E_AxisState.MOVE_ABS://-----------------------------------------------------------------------------------------MOVE_ABS:

							IF posTarget > fPositionLimitMin AND
							   posTarget < fPositionLimitMax
 								THEN 
									bReq_MoveABS := TRUE;
									eState := E_AxisState.MOVING_ABS;
							END_IF
							stY_Axis.bSetToHome			  :=FALSE;
							
							
E_AxisState.MOVING_ABS://-------------------------------------------------------------------------------------MOVING_ABS:

							IF fbMoveABS.Done THEN
									
									bReq_MoveABS := FALSE;
									eState := E_AxisState.IN_TARGET_POS;
									
							ELSIF tonMoveTimeout.Q THEN
									
									bReq_MoveABS := FALSE;
									eState := E_AxisState.ERROR;
							END_IF
							//TO KNOW POSITION OF AXIS
							GVL_HMI.bY_AxisInPosition1		:= FALSE;
							GVL_HMI.bY_AxisInPosition2		:= FALSE;
							GVL_HMI.bY_AxisInPosition3		:= FALSE;
							GVL_HMI.bY_AxisInHomePosition	:= FALSE;

E_AxisState.MOVE_REL:;
E_AxisState.MOVING_REL:;

E_AxisState.IN_TARGET_POS://-------------------------------------------------------------------------------IN_TARGET_POS:

							IF tonActionDone.Q THEN
								eState := E_AxisState.AXIS_READY;
							END_IF
							//TO KNOW THE POSITION OF THE AXIS
							IF stY_Axis.bSetToPosition[1] THEN
								GVL_HMI.bY_AxisInPosition1				:= TRUE;
							END_IF
							IF stY_Axis.bSetToPosition[2] THEN
								GVL_HMI.bY_AxisInPosition2				:= TRUE;
							END_IF
							IF stY_Axis.bSetToPosition[3] THEN
								GVL_HMI.bY_AxisInPosition3				:= TRUE;
							END_IF
							IF stY_Axis.bSetToHome THEN
								GVL_HMI.bY_AxisInHomePosition			:= TRUE;
							END_IF
E_AxisState.ERROR://-----------------------------------------------------------------------------------------------ERROR:

	 					eState := E_AxisState.ABORTED;
						
E_AxisState.MANUAL_MODE://-----------------------------------------------------------------------------------MANUAL_MODE:

							e_Manual();
					
							IF NOT CMD.bManualMode THEN
								eState := E_AxisState.ABORTED;
							END_IF

ELSE 
eState := E_AxisState.ABORTED;
END_CASE //------------------------------------------------------------------------------------------------------END_CASE

(******************************************************STATUS************************************************************)
// Module Status
status.bReady	:= eState = E_AxisState.AXIS_READY;

status.bBusy	:= eState <> E_AxisState.ABORTED	AND
				   eState <> E_AxisState.AXIS_READY AND
				   eState <> E_AxisState.IN_TARGET_POS AND
				   eState <> E_AxisState.ERROR;
				   
status.bDone	:= eState = E_AxisState.IN_TARGET_POS;

status.bError	:= eState = E_AxisState.ERROR OR 
				   fbPower.Error OR fbStop.Error OR fbMoveABS.Error OR fbMoveREL.Error; 
//---------------------------------------------------------------------------------------------------------------oldschoo1
END_ACTION

ACTION b_Call_AxisFBs:
// CTRL FBs Call

	fbPower 	(Axis:=refY_Axis, Enable:=bReq_Power, Enable_Positive:=bReq_Power, Enable_Negative:=bReq_Power);
	fbReset 	(Axis:=refY_Axis, Execute:=bReq_Reset);
	
  fbMoveABS 	(Axis:=refY_Axis, Execute:=bReq_MoveABS, 
				 Position:=posTarget, Velocity:= SEL(bRetract,cfgAxis.fTargetVelocity,cfgAxis.fRetractVelocity));
  fbMoveREL 	(Axis:=refY_Axis, Execute:=FALSE);
 	 fbStop 	(Axis:=refY_Axis, Execute:=FALSE);
  fbReadPos		(Axis:=refY_Axis, Enable:=eState=E_AxisState.HOMING);
fbParameter[0]  (Axis:=refY_Axis, Enable:=TRUE, ParameterNumber:=MC_AXISPARAMETER.AxisMinSoftPosLimit, Value=>fLimitPositionLow);
fbParameter[1]  (Axis:=refY_Axis, Enable:=TRUE, ParameterNumber:=MC_AXISPARAMETER.AxisMaxSoftPosLimit, Value=>fLimitPositionHigh);
fbReadStatus	(Axis:=refY_Axis, Enable:=TRUE, Status=>stAxisStatus, Error=>bAxisInError);
//-----------------------------------------------------------------------------------------------------------------------oldschoo1
END_ACTION

METHOD c_Get_TargetPositon	:LREAL
VAR_INPUT

	// Positions
    posHome     			:LREAL;
    posPoints   			:ARRAY[1..3]OF LREAL;
    fOffsets  				:ARRAY[1..3]OF LREAL;
	
	// Set Target Flags
    bSetHome    			:BOOL;
    bSetPoint   			:ARRAY[1..3]OF BOOL;
	
END_VAR
//----------------------------------------------------------oldschoo1


VAR
	idx           			:INT;
	posTargeteBase	     	:LREAL;
END_VAR
IF bSetHome THEN
    		posTargeteBase := posHome;
ELSE
	
			FOR idx:= 1 TO 3 
			DO
					IF bSetPoint[idx] THEN
						posTargeteBase := posPoints[idx] + fOffsets[idx];
						EXIT;
					END_IF		
			END_FOR
END_IF

c_Get_TargetPositon	:= posTargeteBase;
//--------------------------------------------------------------oldschoo1
END_METHOD

ACTION d_Get_CurrentPosition:
IF fbReadPos.Valid THEN fCurrentPosition:=fbReadPos.Position; END_IF
//----------------------------------------------------------oldschoo1
END_ACTION

ACTION e_Manual:
posTarget := c_Get_TargetPositon(
															posHome 	:= cfgAxis.posHome,
															posPoints   := cfgAxis.posWorkPositions,
															fOffsets	:= fOffsets,
															bSetHome 	:= stY_Axis.bSetToHome,
															bSetPoint 	:= stY_Axis.bSetToPosition
															);	
trigbMoveToPos( CLK := GVL_HMI.bMoveToPos );
IF GVL_HMI.bY_AxisPosition1 THEN
	stY_Axis.bSetToPosition[1]			:= TRUE;
	GVL_HMI.bMoveToPos					:= TRUE;
END_IF
IF GVL_HMI.bY_AxisPosition2 THEN
	stY_Axis.bSetToPosition[2]			:= TRUE;
	GVL_HMI.bMoveToPos					:= TRUE;
END_IF
IF GVL_HMI.bY_AxisPosition3 THEN
	stY_Axis.bSetToPosition[3]			:= TRUE;
	GVL_HMI.bMoveToPos					:= TRUE;
END_IF
IF GVL_HMI.bY_HomePosition THEN
	stY_Axis.bSetToHome					:= TRUE;
	GVL_HMI.bMoveToPos					:= TRUE;
END_IF
	
IF trigbMoveToPos.Q THEN
	nManualModeState					:=10;
END_IF

CASE nManualModeState OF
	
10:
IF posTarget > fPositionLimitMin AND
		posTarget < fPositionLimitMax THEN 
		bReq_MoveABS 					:= TRUE;
		GVL_HMI.bY_AxisInPosition1Man	:= FALSE;
		GVL_HMI.bY_AxisInPosition2Man	:= FALSE;
		GVL_HMI.bY_AxisInPosition3Man	:= FALSE;
		GVL_HMI.bY_AxisInHomePositionMan:= FALSE;
		nManualModeState				:=20;
	END_IF	
20:
IF fbMoveABS.Done THEN	
	IF stY_Axis.bSetToPosition[1] THEN
		GVL_HMI.bY_AxisInPosition1Man	:= TRUE;
	END_IF
	IF stY_Axis.bSetToPosition[2] THEN
		GVL_HMI.bY_AxisInPosition2Man	:= TRUE;
	END_IF
	IF stY_Axis.bSetToPosition[3] THEN
		GVL_HMI.bY_AxisInPosition3Man	:= TRUE;
	END_IF
	IF stY_Axis.bSetToHome THEN
		GVL_HMI.bY_AxisInHomePositionMan:= TRUE;
	END_IF
	nManualModeState					:=30;
END_IF
	
30:								
		bReq_MoveABS 					:= FALSE;
		stY_Axis.bSetToPosition[1]		:= FALSE;
		stY_Axis.bSetToPosition[2]		:= FALSE;
		stY_Axis.bSetToPosition[3]		:= FALSE;
		stY_Axis.bSetToHome				:= FALSE;
		GVL_HMI.bMoveToPos				:= FALSE;
		
IF NOT GVL_Master.stMachineStatus.bManualMode THEN
		GVL_HMI.bY_AxisInPosition1Man	:= FALSE;
		GVL_HMI.bY_AxisInPosition2Man	:= FALSE;
		GVL_HMI.bY_AxisInPosition3Man	:= FALSE;
		GVL_HMI.bY_AxisInHomePositionMan:= FALSE;
END_IF
END_CASE
END_ACTION

END_PROGRAM

// ---- POUs/01_MODULES/KISTLER/K_Master_Kistler.TcPOU
PROGRAM K_Master_Kistler
VAR
	
	bFirstRun							:BOOL:=TRUE;
	
	//Module CTRL
	eState								:E_KistlerState:=E_KistlerState.ENABLE_PLC_CTRL;
	eErrorID							:E_KistlerErrorID;
	
	//Parameters
	fHomePositionTolerance				:REAL:= 1.5;	// > 2mm may cause Pack insertion issues
	fbForceMonitor						:FB_ForceMonitor;
	FBDistanceMonitor					: FB_DistanceMonitor;
	fUVT_00								:REAL;
	fUVT_01								:REAL;	
	fDistanceSetpoint					:REAL;
	//Timers && Triggers
	tonAbortModule						:Tc2_Standard.TON;
	tonResetError						:Tc2_Standard.TON;
	tonEnableDrive						:Tc2_Standard.TON;
	tonActionDone						:Tc2_Standard.TON;
	tonActionTimeout					:Tc2_Standard.TON;
	tonPowerUpTimeout					:Tc2_Standard.TON;	
	tonDelaySignals						:ARRAY[1..11]OF Tc2_Standard.TON;
	
	rcmdbExecute						:R_TRIG;
	
	//EtherCAT - Kistler CTRL
	stSendCMD							:ST_KistlerData_CMD;
	

	//Com Data Proccessing
	stTemp								:ST_KistlerData_Temporary;//Temp. only
	fbUnpack							:ARRAY[0..199]OF FB_UnpackByteToBoolArray;
	fbByte2Real							:FB_ArrayOfByte2Real;
	fbRealPosition2Byte					:FB_Real2ArrayOfByte;
	fbRealSpeed2Byte					:FB_Real2ArrayOfByte;
	fbPositiontosend					:FB_Byte_To_Bits;
	fbSpeedtosend						:FB_Byte_To_Bits;
	
	// Live readings Local
	rKistlerLive_X						:REAL;	//Travel
	rKistlerLive_Y						:REAL;	//Force
	
	// Process Record
	bForceMonitorActive					:BOOL;	//Recording Start/Stop
	
	
	//Support variables
	idx1								:INT;	//indexer
	idx2								:INT;	//indexer
	idx3								:INT;	//indexer
	
	//Manual
	trigCycleMan						:R_TRIG;
	tonRstCycSignalMan					:TON;
	bTest								:BOOL;
	
	rPosition							:FB_BytesToReal;
	rSpeed								:FB_BytesToReal;
	
	bDistancePass						: BOOL;
	bDistanceFail						: BOOL;
	
END_VAR
VAR_OUTPUT
	stKistlerReport						:ST_ProcessReport;
END_VAR


//--------------------IN/OUT-----------------------------------------------------------------*
VAR_INPUT	
	CMD									:ST_ModuleCMD;	
END_VAR
VAR_OUTPUT	
	STATUS								:ST_ModuleStatus;
	stReceived							:ST_KistlerData_Status;	
END_VAR
//-----------------------------------------------------------------------------------oldschoo1

PRG_Fault_Kistler(aAlarms := GVL_Master.stAlarms);
//Call for Actions
a_Unpack_Received();
b_Ctrl_Kistler();
d_Monitor_ProcessForce();
f_Pack_DataToSend();


// Map to HMI
GVL_HMI.rKistlerLiveReading_X		:= rKistlerLive_X;	//Realtime X travel distance
GVL_HMI.rKistlerLiveReading_Y		:= rKistlerLive_Y;	//Realtime Y force reading

fDistanceSetpoint				:= GVL_PERSISTENT.rReservoir_BottomPosition - GVL_PERSISTENT.rReservoir_Bottomlimitoffset;

//--------------------------------------------------------------------------oldschoo1

ACTION a_Unpack_Received:
//Thanks for the Telegram, it's been received:)
FOR idx1:= 0 TO 199 
DO 
fbUnpack[idx1].inputByte := GVL_MODULES.stKistler.st_TelegramDataIn[idx1];
fbUnpack[idx1](outputBits := stTemp.arrInBits[idx1]);
END_FOR
//---------------------------------------------------------------oldschoo1

//  Byte 0  –  Basic CTRL Mirror  ---------------------------------------
stReceived.bStart_Mirror						:= stTemp.arrInBits[0][0];
stReceived.bTareY_Mirror						:= stTemp.arrInBits[0][1];
stReceived.bZeroX_Mirror						:= stTemp.arrInBits[0][2];
stReceived.bSTestX_Mirror						:= stTemp.arrInBits[0][3];
stReceived.bSTestY_Mirror						:= stTemp.arrInBits[0][4];
stReceived.bMasterMeas_Mirror					:= stTemp.arrInBits[0][6];
stReceived.bIncZero_Mirror						:= stTemp.arrInBits[0][7];

//  Byte 1  –  Login Mirror  --------------------------------------------
stReceived.bAckAdminGlobal_Mirror				:= stTemp.arrInBits[1][0];
stReceived.bAckAdmin_Mirror						:= stTemp.arrInBits[1][1];
stReceived.bAccess_Mirror						:= stTemp.arrInBits[1][3];
stReceived.bAuto_Mirror							:= stTemp.arrInBits[1][4];
stReceived.bStatReset_Mirror					:= stTemp.arrInBits[1][5];
stReceived.bStatDisable_Mirror					:= stTemp.arrInBits[1][6];
stReceived.bTareExtY_Mirror						:= stTemp.arrInBits[1][7];

//  Byte 2  –  Measurement Program No. Mirror  --------------------------
stReceived.mpNumber_Mirror[0]					:= stTemp.arrInBits[2][0];
stReceived.mpNumber_Mirror[1]					:= stTemp.arrInBits[2][1];
stReceived.mpNumber_Mirror[2]					:= stTemp.arrInBits[2][2];
stReceived.mpNumber_Mirror[3]					:= stTemp.arrInBits[2][3];
stReceived.mpNumber_Mirror[4]					:= stTemp.arrInBits[2][4];
stReceived.mpNumber_Mirror[5]					:= stTemp.arrInBits[2][5];
stReceived.mpNumber_Mirror[6]					:= stTemp.arrInBits[2][6];

//  Byte 3  –  Service / Brake  -----------------------------------------
stReceived.bResetSNGen_Mirror					:= stTemp.arrInBits[3][2];
stReceived.bBrakeTestActive						:= stTemp.arrInBits[3][5];
stReceived.bExportPvt_Mirror					:= stTemp.arrInBits[3][6];

//  Byte 4  –  Configurable Inputs Mirror  ------------------------------
stReceived.bIUni_Mirror[0]						:= stTemp.arrInBits[4][0];
stReceived.bIUni_Mirror[1]						:= stTemp.arrInBits[4][1];
stReceived.bIUni_Mirror[2]						:= stTemp.arrInBits[4][2];
stReceived.bIUni_Mirror[3]						:= stTemp.arrInBits[4][3];
stReceived.bIUni_Mirror[4]						:= stTemp.arrInBits[4][4];
stReceived.bIUni_Mirror[5]						:= stTemp.arrInBits[4][5];
stReceived.bIUni_Mirror[6]						:= stTemp.arrInBits[4][6];
stReceived.bIUni_Mirror[7]						:= stTemp.arrInBits[4][7];

//  Byte 6  –  Global Status  -------------------------------------------
stReceived.bReady								:= stTemp.arrInBits[6][0];
stReceived.bOkTotal								:= stTemp.arrInBits[6][1];
stReceived.bNokTotal							:= stTemp.arrInBits[6][2];
stReceived.bNoPass								:= stTemp.arrInBits[6][3];
stReceived.bWarning								:= stTemp.arrInBits[6][6];
stReceived.bAlarm								:= stTemp.arrInBits[6][7];

//  Byte 7  –  Switching Signals  ---------------------------------------
stReceived.bS1									:= stTemp.arrInBits[7][0];
stReceived.bS2									:= stTemp.arrInBits[7][1];

//  Byte 8  –  O_UNI  ---------------------------------------------------
stReceived.bO_UNI[0]							:= stTemp.arrInBits[8][0];
stReceived.bO_UNI[1]							:= stTemp.arrInBits[8][1];

//  Byte 9  –  Drive / Sequence Mirror  ---------------------------------
stReceived.bDriveEnable_Mirror					:= stTemp.arrInBits[9][0];
stReceived.bRunSequence_Mirror					:= stTemp.arrInBits[9][1];
stReceived.bDriveHome_Mirror					:= stTemp.arrInBits[9][2];
stReceived.bDriveRef_Mirror						:= stTemp.arrInBits[9][3];
stReceived.bJogFwd_Mirror						:= stTemp.arrInBits[9][4];
stReceived.bJogBack_Mirror						:= stTemp.arrInBits[9][5];
stReceived.bWaitRequest							:= stTemp.arrInBits[9][6];
stReceived.bBrakeTestDone						:= stTemp.arrInBits[9][7];

//  Byte 10 –  Sequence State  -------------------------------------------
stReceived.bSeqStopped							:= stTemp.arrInBits[10][0];
stReceived.bSeqEnd								:= stTemp.arrInBits[10][1];
stReceived.bOnlineEoNok							:= stTemp.arrInBits[10][2];
stReceived.bSeqExtStop							:= stTemp.arrInBits[10][3];
stReceived.bSeqError							:= stTemp.arrInBits[10][4];
stReceived.bDriveEnabled						:= stTemp.arrInBits[10][5];
stReceived.bHomePosReached						:= stTemp.arrInBits[10][6];
stReceived.bRefPosReached						:= stTemp.arrInBits[10][7];

//  Byte 11 –  Servo / Safety  -------------------------------------------
stReceived.bStandstill							:= stTemp.arrInBits[11][0];
stReceived.bBrakeTestReq						:= stTemp.arrInBits[11][1];
stReceived.bServoWarn							:= stTemp.arrInBits[11][2];
stReceived.bServoError							:= stTemp.arrInBits[11][3];
stReceived.bSMES_Or_STO							:= stTemp.arrInBits[11][4];
stReceived.bSMST2								:= stTemp.arrInBits[11][5];
stReceived.bSMM1								:= stTemp.arrInBits[11][6];
stReceived.bUserModeActive						:= stTemp.arrInBits[11][7];

//  Byte 12 –  Current Sequence Mirror  ----------------------------------
stReceived.bCurrSeqMain_Mirror					:= stTemp.arrInBits[12][0];
stReceived.bCurrSeqSub_Mirror					:= stTemp.arrInBits[12][1];

//  Byte 19 –  Device / Transfer Flags  ----------------------------------
stReceived.bTransmissionFault					:= stTemp.arrInBits[19][0];
stReceived.bAck									:= stTemp.arrInBits[19][1];
stReceived.bDeviceAvailable						:= stTemp.arrInBits[19][2];
stReceived.bMpChanged							:= stTemp.arrInBits[19][4];
stReceived.bGlobalChanged						:= stTemp.arrInBits[19][6];
stReceived.bBackupComplete						:= stTemp.arrInBits[19][7];

(************************************Payload**************************************)
//  Bytes 20-27 –  Live XY values  ----------------------------------------------*
FOR idx3:= 20 TO 23					
DO
stReceived.pvCurrentValueX[idx3] := FUN_PackBoolArrayToByte(stTemp.arrInBits[idx3]);
																		    END_FOR
							     fbByte2Real.arrBytes := stReceived.pvCurrentValueX;
							     fbByte2Real();rKistlerLive_X := fbByte2Real.rValue;
																			
FOR idx3:= 24 TO 27					
DO
stReceived.pvCurrentValueY[idx3] := FUN_PackBoolArrayToByte(stTemp.arrInBits[idx3]);
																			END_FOR
							     fbByte2Real.arrBytes := stReceived.pvCurrentValueY;
							     fbByte2Real();rKistlerLive_Y := fbByte2Real.rValue;
//--------------------------------------------------------------------------oldschoo1

rPosition(inBytes:= , outReal=> );
rSpeed(inBytes:= , outReal=> );
END_ACTION

ACTION b_Ctrl_Kistler:
// Timmers && Triggers
tonActionDone     (IN:= FALSE,
			       PT:= T#100MS);
tonActionTimeout  (IN:= eState=E_KistlerState.WAIT_CYCLE_DONE,
			       PT:= T#90S);
tonPowerUpTimeout (IN:= eState=E_KistlerState.ENABLE_DRIVE,
				   PT:=T#20S);				   
tonResetError     (IN:= stReceived.bServoError OR stReceived.bAlarm,
			       PT:= T#500MS);
tonAbortModule	  (IN:= cmd.bAbort OR (NOT stSafety.bSafety_OK) OR (NOT cmd.bEnable),
				   PT:= T#100MS);
				   
//Signal pulses && delays				  
tonDelaySignals[1](IN:= eState=E_KistlerState.ENABLE_PLC_CTRL AND stSendCMD.bAckAdminGlobal,
				   PT:= T#100MS);
tonDelaySignals[2](IN:= eState=E_KistlerState.RESET_ERROR AND (stReceived.bAlarm OR stReceived.bServoError) AND NOT tonDelaySignals[3].Q,
				   PT:= T#1S);
tonDelaySignals[3](IN:= eState=E_KistlerState.RESET_ERROR AND stSendCMD.bAckAdmin,
				   PT:= T#1S);
tonDelaySignals[4](IN:= eState=E_KistlerState.ENABLE_DRIVE,
				   PT:= T#100MS);
tonDelaySignals[5](IN:= eState=E_KistlerState.SET_PARAMETERS,
				   PT:=T#330MS);
tonDelaySignals[6](IN:=eState=E_KistlerState.RECORD_CYCLE_DATA, 
				   PT:=T#50MS);				   
tonDelaySignals[7](IN:=eState=E_KistlerState.ERROR, 
				   PT:=T#330MS);
tonDelaySignals[8](IN:=eState=E_KistlerState.PRESS_CYCLE, 
				   PT:=T#330MS);
tonDelaySignals[9](IN:=eState=E_KistlerState.GOTO_HOME_POS, 
				   PT:=T#330MS);
tonDelaySignals[10](IN:=eState=E_KistlerState.SET_PARAMETERS AND stReceived.bTareY_Mirror AND tonDelaySignals[5].Q, 
				   PT:=T#3S);
tonDelaySignals[11]( IN := NOT stReceived.bAlarm, PT := T#1S);

rcmdbExecute( CLK := cmd.bExecute);
(*****************************************************RESET**********************************************************)
// Reset Errors
(*IF cmd.bReset OR tonResetError.Q THEN
 			  
			status.bError 	:= TRUE;
            eState := E_KistlerState.RESET_ERROR;
			END_IF*)

// Abort Action
IF tonAbortModule.q THEN
	
			stSendCMD.bDriveEnable	:= FALSE;
			stSendCMD.bAckAdmin		:= FALSE;
			stSendCMD.bDriveToRef	:= FALSE;
			stSendCMD.bTareY 		:= FALSE;
			stSendCMD.bRunSequence  := FALSE;
			eState := E_KistlerState.ABORTED;
			END_IF	
(*******************************************************CTRL**********************************************************)
IF CMD.bManualMode THEN
	eState := E_KistlerState.MANUAL;
END_IF
// Kistler CTRL State Machine
CASE eState OF //-----------------------------------------------------------------------------------------------------SM

E_KistlerState.ENABLE_PLC_CTRL://-----------------------------------------------------------------------ENABLE_PLC_CTRL:

						IF stReceived.bReady AND NOT bSystemPoweringUP THEN
								stSendCMD.bAuto:=TRUE; 
						ELSIF NOT stReceived.bReady THEN
								status.nErrorID:= TO_INT(eErrorID=E_KistlerErrorID.COMUNICATION_ERROR);
						END_IF
								
						IF stReceived.bAuto_Mirror THEN
								stSendCMD.bAckAdminGlobal:=TRUE;
						END_IF
						IF tonDelaySignals[1].Q THEN
 								stSendCMD.bAckAdminGlobal:=FALSE;
								eState := E_KistlerState.ABORTED;
								END_IF

E_KistlerState.ABORTED://---------------------------------------------------------------------------------------ABORTED:
					
						IF (NOT stReceived.bAuto_Mirror) AND 
						   (NOT cmd.bAbort) AND stSafety.bSafety_OK AND cmd.bEnable THEN
								eState := E_KistlerState.ENABLE_PLC_CTRL;
							
						ELSIF stReceived.bAuto_Mirror AND 
							 (NOT cmd.bAbort) AND stSafety.bSafety_OK AND cmd.bEnable THEN
								eState := E_KistlerState.ENABLE_DRIVE;
						END_IF
								

E_KistlerState.ENABLE_DRIVE://-----------------------------------------------------------------------------ENABLE_DRIVE:
	
						c_Select_Program();

						IF tonDelaySignals[4].Q THEN
								stSendCMD.bDriveEnable:=TRUE; END_IF
						
						IF stReceived.bDriveEnabled THEN
								eState := E_KistlerState.RESET_ERROR;
								
						ELSIF (NOT stReceived.bDriveEnabled) AND tonPowerUpTimeout.Q THEN
								status.nErrorID:= TO_INT(eErrorID=E_KistlerErrorID.ENABLE_DRIVE_ERROR);
								eState := E_KistlerState.ERROR;
						END_IF

E_KistlerState.RESET_ERROR://-------------------------------------------------------------------------------RESET_ERROR:
					
						IF stReceived.bAlarm OR stReceived.bServoError  THEN
								IF tonDelaySignals[2].Q THEN
								stSendCMD.bAckAdmin:=TRUE; END_IF
						END_IF
		
						IF tonDelaySignals[3].Q THEN
								stSendCMD.bAckAdmin:=FALSE; END_IF
								
						IF (tonDelaySignals[11].Q) AND (NOT stReceived.bServoError) THEN
								stSendCMD.bAckAdmin:=FALSE;
								status.nErrorID:= TO_INT(eErrorID=E_KistlerErrorID.NO_ERROR);
								eState := E_KistlerState.GOTO_HOME_POS;
						END_IF
						
E_KistlerState.GOTO_HOME_POS://---------------------------------------------------------------------------GOTO_HOME_POS:

						IF NOT stReceived.bHomePosReached AND stReceived.bReady AND
								tonDelaySignals[9].Q THEN

								stSendCMD.bDriveToRef:= TRUE;
						END_IF
						
						IF stReceived.bHomePosReached OR rKistlerLive_X < fHomePositionTolerance THEN

								stSendCMD.bDriveToRef:= FALSE;
								eState := E_KistlerState.SET_PARAMETERS;
						END_IF
	
E_KistlerState.SET_PARAMETERS://-------------------------------------------------------------------------SET_PARAMETERS:

						stSendCMD.bTareY := TRUE;
						fUVT_00:= GVL_PERSISTENT.rReservoir_BottomPosition;
						fUVT_01:= GVL_PERSISTENT.rKistlerForce_Speed;
						
						IF stReceived.bTareY_Mirror AND tonDelaySignals[5].Q THEN
								stSendCMD.bTareY := FALSE;
								eState := E_KistlerState.PRESS_READY;
						END_IF

E_KistlerState.PRESS_READY://-------------------------------------------------------------------------------PRESS_READY:

						IF stReceived.bReady AND rcmdbExecute.Q THEN
								eState := E_KistlerState.PRESS_CYCLE;
						END_IF

						
E_KistlerState.PRESS_CYCLE://-------------------------------------------------------------------------------PRESS_CYCLE:


						stSendCMD.bRunSequence := TRUE;
						
						IF stReceived.bRunSequence_Mirror  AND tonDelaySignals[8].Q THEN
								eState := E_KistlerState.WAIT_CYCLE_DONE;
						END_IF
						
E_KistlerState.WAIT_CYCLE_DONE://-----------------------------------------------------------------------WAIT_PRESS_DONE:
						
						IF stReceived.bSeqEnd AND NOT stReceived.bSeqError THEN

								stSendCMD.bRunSequence := FALSE;	
								eState := E_KistlerState.RECORD_CYCLE_DATA;
						
						ELSIF stReceived.bSeqError THEN
								status.nErrorID:= TO_INT(eErrorID=E_KistlerErrorID.PROCESS_ERROR);
								eState := E_KistlerState.ERROR;
	
						ELSIF tonActionTimeout.Q THEN
								status.nErrorID:= TO_INT(eErrorID=E_KistlerErrorID.ACTION_TIMEOUT_ERROR);
								eState := E_KistlerState.ERROR;		
						END_IF
					
E_KistlerState.RECORD_CYCLE_DATA://-------------------------------------------------------------------RECORD_CYCLE_DATA:

			 			

			stKistlerReport.bKis_Pass := fbForceMonitor.bPass AND bDistancePass;
			stKistlerReport.bKis_Fail := fbForceMonitor.bFail OR bDistanceFail;
			stKistlerReport.rKis_HighestRecordedForce := fbForceMonitor.fHighestRecordedForce;
			stKistlerReport.rKis_LowestRecordedForce := fbForceMonitor.fLowestRecordedForce;
			stKistlerReport.rKis_DistanceRecord:=FBDistanceMonitor.MaxDistance;
			stKistlerReport.rKis_Settings_ForceUPPERtreshold := GVL_PERSISTENT.rKistlerForce_UpperLimit;
			stKistlerReport.rKis_Settings_ForceLOWERtreshold := GVL_PERSISTENT.rKistlerForce_LowerLimit;
			stKistlerReport.rKis_Settings_StartMeasurePoint := GVL_PERSISTENT.rReservoir_ContactPosition;
			stKistlerReport.rKis_Settings_ReservoirBottomPoint := GVL_PERSISTENT.rReservoir_BottomPosition;
			
						IF tonDelaySignals[6].Q THEN
								eState := E_KistlerState.PRESS_READY; END_IF	
				
E_KistlerState.JOG_MODE:;
E_KistlerState.ERROR://-------------------------------------------------------------------------------------------ERROR:
						stSendCMD.bDriveEnable	:= FALSE;
						stSendCMD.bAckAdmin		:= FALSE;
						stSendCMD.bDriveToRef	:= FALSE;
						stSendCMD.bTareY 		:= FALSE;
						stSendCMD.bRunSequence  := FALSE;
						
						IF tonDelaySignals[7].Q THEN
					 			eState := E_KistlerState.ABORTED; END_IF
E_KistlerState.MANUAL:
						g_Manual();
						IF NOT CMD.bManualMode THEN
							eState := E_KistlerState.ABORTED;
						END_IF
								
ELSE 
eState := E_KistlerState.ABORTED;
END_CASE //-----------------------------------------------------------------------------------------------------END_CASE

// -------------------------------------------HMI Show Record -------------------------------------------------------//
				IF 	eState = E_KistlerState.PRESS_READY AND (stKistlerReport.bKis_Pass OR stKistlerReport.bKis_Fail) THEN 
					
					GVL_HMI.rKisterldistanceHMI:= FBDistanceMonitor.MaxDistance;
					GVL_HMI.rKisterlForceHMI:=stKistlerReport.rKis_HighestRecordedForce;
					ELSE 
						GVL_HMI.rKisterldistanceHMI:= GVL_HMI.rKistlerLiveReading_X;
						GVL_HMI.rKisterlForceHMI:= GVL_HMI.rKistlerLiveReading_Y;
					END_IF


(******************************************************STATUS***********************************************************)
// Module Status
status.bReady				:= eState = E_KistlerState.PRESS_READY AND 
							   			stReceived.bReady;

status.bBusy				:= eState <> E_KistlerState.ABORTED		AND
				   			   eState <> E_KistlerState.PRESS_READY AND
				   			   eState <> E_KistlerState.ERROR;
				   
status.bActionInProggress	:= eState = E_KistlerState.PRESS_CYCLE OR
				   			   eState = E_KistlerState.WAIT_CYCLE_DONE OR
							   eState = E_KistlerState.RECORD_CYCLE_DATA;
							   
status.bDone				:= eState = E_KistlerState.RECORD_CYCLE_DATA;

status.bError				:= eState = E_KistlerState.ERROR OR 
				   			   stReceived.bServoError; 				 
//-------------------------------------------------------------------------------------------------------------oldschoo1
END_ACTION

ACTION c_Select_Program:
// MP No.selection is 6-bits binary
stSendCMD.mpNumber[0]:=1;  
stSendCMD.mpNumber[1]:=1;  
stSendCMD.mpNumber[2]:=0;  
stSendCMD.mpNumber[3]:=0;  
stSendCMD.mpNumber[4]:=0;  
stSendCMD.mpNumber[5]:=0;  
stSendCMD.mpNumber[6]:=0; 
//------------------------oldschoo1
END_ACTION

ACTION d_Monitor_ProcessForce:

//Trigger
bForceMonitorActive := (eState=E_KistlerState.PRESS_CYCLE OR eState=E_KistlerState.WAIT_CYCLE_DONE);(*AND 
					   (rKistlerLive_X > GVL_PERSISTENT.rReservoir_ContactPosition AND
						rKistlerLive_X < GVL_PERSISTENT.rReservoir_BottomPosition) AND stReceived.bO_UNI[0]*);

//Monitor
fbForceMonitor(
				bEnable := eState=E_KistlerState.PRESS_CYCLE OR eState=E_KistlerState.WAIT_CYCLE_DONE
							OR eState = E_KistlerState.RECORD_CYCLE_DATA,//stReceived.bAuto_Mirror,
				bActive := bForceMonitorActive,
				bReset	:= eState=E_KistlerState.PRESS_READY OR 
						   eState=E_KistlerState.ERROR OR cmd.bReset,
				fDistanceSetpoint := fDistanceSetpoint,
				fDistance := rKistlerLive_X,
 
				fForceInput 		  := rKistlerLive_Y,
				bPass				  =>,
				bFail				  =>,
				fHighestRecordedForce =>,
				fLowestRecordedForce  =>,
				fThreshold_UpperLimit := GVL_PERSISTENT.rKistlerForce_UpperLimit,
				fThreshold_LowerLimit := GVL_PERSISTENT.rKistlerForce_LowerLimit,
				fDebounceTolerance	  := GVL_PERSISTENT.rMeasurementTolerance );
				
//------------------------------------------------------------------------------------------------oldschoo1


FBDistanceMonitor(
	StartSignal:= eState=E_KistlerState.PRESS_CYCLE , 
	EndSignal:= stReceived.bSeqEnd,//eState=E_KistlerState.PRESS_READY, 
	DistanceMaxSetpoint:= , 
	DistanceInput:= rKistlerLive_X,
	fDistanceSetpoint := fDistanceSetpoint, 
	MaxDistance=> , 
	IsMeasuring=>,
	bDistancePass =>bDistancePass,
	bDistanceFail => bDistanceFail);
END_ACTION

ACTION f_Pack_DataToSend:
//  Byte 0  –  Basic CTRL  ----------------------------------------------*
stTemp.arrOutBits[0][0] 					:= stSendCMD.bStart;
stTemp.arrOutBits[0][1] 					:= stSendCMD.bTareY;
											   stSendCMD.bZeroX:=0; //Carefull, Teach Global 0 Position!!!
stTemp.arrOutBits[0][2] 					:= stSendCMD.bZeroX;//*
stTemp.arrOutBits[0][3] 					:= stSendCMD.bSTestX;
stTemp.arrOutBits[0][4] 					:= stSendCMD.bSTestY;
stTemp.arrOutBits[0][5] 					:= 0;
stTemp.arrOutBits[0][6] 					:= stSendCMD.bMasterMeas;
stTemp.arrOutBits[0][7] 					:= stSendCMD.bIncZero;
//  Byte 1  –  Login / Mode  ---------------------------------------------*
stTemp.arrOutBits[1][0] 					:= stSendCMD.bAckAdminGlobal;
stTemp.arrOutBits[1][1] 					:= stSendCMD.bAckAdmin;
stTemp.arrOutBits[1][2] 					:= 0;
stTemp.arrOutBits[1][3] 					:= stSendCMD.bAccess;
stTemp.arrOutBits[1][4] 					:= stSendCMD.bAuto;		//Set false to use TeachingPendant
stTemp.arrOutBits[1][5] 					:= stSendCMD.bStatReset;
stTemp.arrOutBits[1][6] 					:= stSendCMD.bStatDisable;
stTemp.arrOutBits[1][7] 					:= stSendCMD.bTareExtY;
//  Byte 2  –  Measurement Program No.  ----------------------------------*
stTemp.arrOutBits[2][0] 					:= stSendCMD.mpNumber[0];  
stTemp.arrOutBits[2][1] 					:= stSendCMD.mpNumber[1];
stTemp.arrOutBits[2][2] 					:= stSendCMD.mpNumber[2];
stTemp.arrOutBits[2][3] 					:= stSendCMD.mpNumber[3];
stTemp.arrOutBits[2][4] 					:= stSendCMD.mpNumber[4];
stTemp.arrOutBits[2][5] 					:= stSendCMD.mpNumber[5];
stTemp.arrOutBits[2][6] 					:= stSendCMD.mpNumber[6];
stTemp.arrOutBits[2][7] 					:= 0;  
 
//	Bytes - 3,4,5,6,7,8//Reserved  ---------------------------------------*
FOR idx1:= 3 TO 8 
DO
	FOR idx2:= 0 TO 7 
	DO
    stTemp.arrOutBits[idx1][idx2]:=FALSE;END_FOR END_FOR

//  Byte 9  –  Drive CTRL  -----------------------------------------------*
stTemp.arrOutBits[9][0] 					:= stSendCMD.bDriveEnable;
stTemp.arrOutBits[9][1] 					:= stSendCMD.bRunSequence;
stTemp.arrOutBits[9][2] 					:= stSendCMD.bDriveToHome;
stTemp.arrOutBits[9][3] 					:= stSendCMD.bDriveToRef;
stTemp.arrOutBits[9][4] 					:= stSendCMD.bJogFwd;
stTemp.arrOutBits[9][5] 					:= stSendCMD.bJogBack;
stTemp.arrOutBits[9][6] 					:= stSendCMD.bContinueWait;
stTemp.arrOutBits[9][7] 					:= stSendCMD.bBrakeTest;
//  Byte 10  –  Extended Stop  -------------------------------------------*
stTemp.arrOutBits[10][0] 					:= 0;
stTemp.arrOutBits[10][1] 					:= 0;
stTemp.arrOutBits[10][2] 					:= 0;
stTemp.arrOutBits[10][3] 					:= stSendCMD.bSeqExtStopReq;
stTemp.arrOutBits[10][4] 					:= 0;
stTemp.arrOutBits[10][5] 					:= 0;
stTemp.arrOutBits[10][6] 					:= 0;
stTemp.arrOutBits[10][7] 					:= 0;

// Byte - 11 // Reserved_2  ----------------------------------------------*
FOR idx3:= 0 TO 7 
DO
   stTemp.arrOutBits[11][idx3]:=FALSE;END_FOR

//  Byte 12  –  Sequence Flags  ------------------------------------------*
stTemp.arrOutBits[12][0] 					:= stSendCMD.bCurrSeqMain;
stTemp.arrOutBits[12][1] 					:= stSendCMD.bCurrSeqSub;
stTemp.arrOutBits[12][2] 					:= 0;
stTemp.arrOutBits[12][3] 					:= 0;
stTemp.arrOutBits[12][4] 					:= 0;
stTemp.arrOutBits[12][5] 					:= 0;
stTemp.arrOutBits[12][6] 					:= 0;
stTemp.arrOutBits[12][7] 					:= 0;

// Byte - 13 // Reserved_3  ----------------------------------------------*
FOR idx3:= 0 TO 7 
DO
   stTemp.arrOutBits[13][idx3]:=FALSE;END_FOR

//  Byte 14  –  Page CTRL (CFG-MP)  --------------------------------------*
stTemp.arrOutBits[14][0] 					:= stSendCMD.mpNumber[0];
stTemp.arrOutBits[14][1] 					:= stSendCMD.mpNumber[1];
stTemp.arrOutBits[14][2] 					:= stSendCMD.mpNumber[2];
stTemp.arrOutBits[14][3] 					:= stSendCMD.mpNumber[3];
stTemp.arrOutBits[14][4] 					:= stSendCMD.mpNumber[4];
stTemp.arrOutBits[14][5] 					:= stSendCMD.mpNumber[5];
stTemp.arrOutBits[14][6] 					:= stSendCMD.mpNumber[6];
stTemp.arrOutBits[14][7] 					:= 0;
// Byte - 15 // Reserved_4  ----------------------------------------------*
FOR idx3:= 0 TO 7 
DO
   stTemp.arrOutBits[15][idx3]:=FALSE;END_FOR
   
//  Byte 16  –  CFG-Address  ---------------------------------------------*
stTemp.arrOutBits[16][0] 					:= 0;
stTemp.arrOutBits[16][1] 					:= 0;
stTemp.arrOutBits[16][2] 					:= 0;
stTemp.arrOutBits[16][3] 					:= 0;
stTemp.arrOutBits[16][4] 					:= 0;
stTemp.arrOutBits[16][5] 					:= 0;
stTemp.arrOutBits[16][6] 					:= 0;
stTemp.arrOutBits[16][7] 					:= 0;
//  Byte 17  –  CFG-Lenght  ----------------------------------------------*
stTemp.arrOutBits[17][0] 					:= 0;
stTemp.arrOutBits[17][1] 					:= 0;
stTemp.arrOutBits[17][2] 					:= 0;
stTemp.arrOutBits[17][3] 					:= 0;
stTemp.arrOutBits[17][4] 					:= 1;
stTemp.arrOutBits[17][5] 					:= 0;
stTemp.arrOutBits[17][6] 					:= 0;
stTemp.arrOutBits[17][7] 					:= 1;
//  Byte 18  –  Select Page  ---------------------------------------------*
stTemp.arrOutBits[18][0] 					:= 0;
stTemp.arrOutBits[18][1] 					:= 0;
stTemp.arrOutBits[18][2] 					:= 0;
stTemp.arrOutBits[18][3] 					:= 0;
stTemp.arrOutBits[18][4] 					:= 0;
stTemp.arrOutBits[18][5] 					:= 0;
stTemp.arrOutBits[18][6] 					:= 0;
stTemp.arrOutBits[18][7] 					:= 0;
//  Byte 19  –  Save / Strobe / Backup  ----------------------------------*
stTemp.arrOutBits[19][0] 					:= 1;
stTemp.arrOutBits[19][1] 					:= bFlash250Hz;
stTemp.arrOutBits[19][2] 					:= 0;
stTemp.arrOutBits[19][3] 					:= 0;
stTemp.arrOutBits[19][4] 					:= 0;
stTemp.arrOutBits[19][5] 					:= 0;
stTemp.arrOutBits[19][6] 					:= 0;
stTemp.arrOutBits[19][7] 					:= 0;

(******************************************Payload**********************************************)
// Byte 136 - 139 - pMeasureTravelBottom  -----------------------------------------------------*

(*Position*)
stTemp.arrOutBits[36][0]:=fbPositiontosend.Result[0];
stTemp.arrOutBits[36][1]:=fbPositiontosend.Result[1];
stTemp.arrOutBits[36][2]:=fbPositiontosend.Result[2];
stTemp.arrOutBits[36][3]:=fbPositiontosend.Result[3];
stTemp.arrOutBits[36][4]:=fbPositiontosend.Result[4];
stTemp.arrOutBits[36][5]:=fbPositiontosend.Result[5];
stTemp.arrOutBits[36][6]:=fbPositiontosend.Result[6];
stTemp.arrOutBits[36][7]:=fbPositiontosend.Result[7];
stTemp.arrOutBits[37][0]:=fbPositiontosend.Result[8];
stTemp.arrOutBits[37][1]:=fbPositiontosend.Result[9];
stTemp.arrOutBits[37][2]:=fbPositiontosend.Result[10];
stTemp.arrOutBits[37][3]:=fbPositiontosend.Result[11];
stTemp.arrOutBits[37][4]:=fbPositiontosend.Result[12];
stTemp.arrOutBits[37][5]:=fbPositiontosend.Result[13];
stTemp.arrOutBits[37][6]:=fbPositiontosend.Result[14];
stTemp.arrOutBits[37][7]:=fbPositiontosend.Result[15];
stTemp.arrOutBits[38][0]:=fbPositiontosend.Result[16];
stTemp.arrOutBits[38][1]:=fbPositiontosend.Result[17];
stTemp.arrOutBits[38][2]:=fbPositiontosend.Result[18];
stTemp.arrOutBits[38][3]:=fbPositiontosend.Result[19];
stTemp.arrOutBits[38][4]:=fbPositiontosend.Result[20];
stTemp.arrOutBits[38][5]:=fbPositiontosend.Result[21];
stTemp.arrOutBits[38][6]:=fbPositiontosend.Result[22];
stTemp.arrOutBits[38][7]:=fbPositiontosend.Result[23];
stTemp.arrOutBits[39][0]:=fbPositiontosend.Result[24];
stTemp.arrOutBits[39][1]:=fbPositiontosend.Result[25];
stTemp.arrOutBits[39][2]:=fbPositiontosend.Result[26];
stTemp.arrOutBits[39][3]:=fbPositiontosend.Result[27];
stTemp.arrOutBits[39][4]:=fbPositiontosend.Result[28];
stTemp.arrOutBits[39][5]:=fbPositiontosend.Result[29];
stTemp.arrOutBits[39][6]:=fbPositiontosend.Result[30];
stTemp.arrOutBits[39][7]:=fbPositiontosend.Result[31];

(*Speed*)
stTemp.arrOutBits[40][0]:=fbSpeedtosend.Result[0];
stTemp.arrOutBits[40][1]:=fbSpeedtosend.Result[1];
stTemp.arrOutBits[40][2]:=fbSpeedtosend.Result[2];
stTemp.arrOutBits[40][3]:=fbSpeedtosend.Result[3];
stTemp.arrOutBits[40][4]:=fbSpeedtosend.Result[4];
stTemp.arrOutBits[40][5]:=fbSpeedtosend.Result[5];
stTemp.arrOutBits[40][6]:=fbSpeedtosend.Result[6];
stTemp.arrOutBits[40][7]:=fbSpeedtosend.Result[7];
stTemp.arrOutBits[41][0]:=fbSpeedtosend.Result[8];
stTemp.arrOutBits[41][1]:=fbSpeedtosend.Result[9];
stTemp.arrOutBits[41][2]:=fbSpeedtosend.Result[10];
stTemp.arrOutBits[41][3]:=fbSpeedtosend.Result[11];
stTemp.arrOutBits[41][4]:=fbSpeedtosend.Result[12];
stTemp.arrOutBits[41][5]:=fbSpeedtosend.Result[13];
stTemp.arrOutBits[41][6]:=fbSpeedtosend.Result[14];
stTemp.arrOutBits[41][7]:=fbSpeedtosend.Result[15];
stTemp.arrOutBits[42][0]:=fbSpeedtosend.Result[16];
stTemp.arrOutBits[42][1]:=fbSpeedtosend.Result[17];
stTemp.arrOutBits[42][2]:=fbSpeedtosend.Result[18];
stTemp.arrOutBits[42][3]:=fbSpeedtosend.Result[19];
stTemp.arrOutBits[42][4]:=fbSpeedtosend.Result[20];
stTemp.arrOutBits[42][5]:=fbSpeedtosend.Result[21];
stTemp.arrOutBits[42][6]:=fbSpeedtosend.Result[22];
stTemp.arrOutBits[42][7]:=fbSpeedtosend.Result[23];
stTemp.arrOutBits[43][0]:=fbSpeedtosend.Result[24];
stTemp.arrOutBits[43][1]:=fbSpeedtosend.Result[25];
stTemp.arrOutBits[43][2]:=fbSpeedtosend.Result[26];
stTemp.arrOutBits[43][3]:=fbSpeedtosend.Result[27];
stTemp.arrOutBits[43][4]:=fbSpeedtosend.Result[28];
stTemp.arrOutBits[43][5]:=fbSpeedtosend.Result[29];
stTemp.arrOutBits[43][6]:=fbSpeedtosend.Result[30];
stTemp.arrOutBits[43][7]:=fbSpeedtosend.Result[31];



fbRealPosition2Byte(rValue:=fUVT_00);
fbRealSpeed2Byte(rValue:=fUVT_01);
fbPositiontosend(fbReal2Byte:=fbRealPosition2Byte.arrBytes );
fbSpeedtosend(fbReal2Byte:=fbRealSpeed2Byte.arrBytes );


(*
//fbReal2Byte(rValue:=fUVT_00);
FOR idx1 := 0 TO 3 
DO
    FOR idx2 := 0 TO 7 
	DO
    stTemp.arrOutBits[136 + idx1][idx2]:=((fbRealPosition2Byte.arrBytes[idx1] AND SHL(1, idx2))<>0);
    	 stTemp.arrOutBits[140 + idx1][idx2]:=((fbRealSpeed2Byte.arrBytes[idx1] AND SHL(1, idx2))<>0);																			
																									END_FOR
END_FOR
*)

(****************************************Pack to Telegram****************************************)
FOR idx3:= 0 TO 199//							|
DO
GVL_MODULES.stKistler.st_TelegramDataOut[idx3] := FUN_PackBoolArrayToByte(stTemp.arrOutBits[idx3]);
																							END_FOR
																		
//-----------------------------------------------------------------------------------------oldschoo1
END_ACTION

ACTION g_Manual:

trigCycleMan( CLK := GVL_HMI.bKistlerCycle );
tonRstCycSignalMan( IN := stSendCMD.bRunSequence, PT := T#500MS);
IF trigCycleMan.Q THEN	
	stSendCMD.bRunSequence := TRUE;
ELSIF stReceived.bSeqEnd AND tonRstCycSignalMan.Q THEN
	stSendCMD.bRunSequence := FALSE;
END_IF
END_ACTION

END_PROGRAM

// ---- POUs/03_Utilities/FB_ForceMonitor.TcPOU
FUNCTION_BLOCK FB_ForceMonitor

VAR_INPUT
	
	//Input parameters
    bEnable                  			:BOOL;   
    bActive                 			:BOOL;	//Monitoring active
	bReset								:BOOL;
    fForceInput              			:REAL;
    fThreshold_UpperLimit    			:REAL;
    fThreshold_LowerLimit   			:REAL;
	fDebounceTolerance   				:REAL;	// +/- range for stable
	fDistance							:REAL;
	fDisTanceSetPoint					:REAL;



END_VAR

VAR_OUTPUT
	
	//Output parameters
    bPass                  			    :BOOL;    //TRUE when within both limits
    bFail                    			:BOOL;    //TRUE if outside
    fHighestRecordedForce    			:REAL;
    fLowestRecordedForce     			:REAL;
    bOutOfRangeHigh          			:BOOL;
    bOutOfRangeLow           			:BOOL;
END_VAR

VAR
	//Debounce
	fForceInputABS						:REAL;

	tDebouncePeriod      				:TIME:= T#75MS;
	tonDebounce      					:Tc2_Standard.TON;
	fForceLastStable     				:REAL;
	fForceFiltered       				:REAL;
	bForceStable         				:BOOL;
	
	bDistancePass						:BOOL;
	//Logic support variables
    bActiveLast              			:BOOL;
    bEvaluate	             			:BOOL;
    bTracking                			:BOOL;
END_VAR

//----------------------------------------------------------------------oldschoo1

//Input ABS
IF fForceInput > 0 THEN      //Correct the error in negative read
fForceInputABS :=ABS(fForceInput);
ELSE 
	fForceInputABS:=0;
END_IF

// Transitions
bEvaluate 	:= NOT bActive AND bActiveLast;
bActiveLast := bActive;


// Debounce logic --------------------------------------------------------------*
IF (fForceInputABS - fForceLastStable) <= fDebounceTolerance THEN
    	tonDebounce(IN:=TRUE, PT:=tDebouncePeriod);
ELSE
    	tonDebounce(IN:=FALSE);
    	fForceLastStable:= fForceInputABS;
END_IF;

bForceStable := tonDebounce.Q;

IF bForceStable THEN fForceFiltered := fForceLastStable; END_IF


// LOGIC ------------------------------------------------------------------------*
IF bEnable  THEN

	//Record
    IF bActive THEN
					IF NOT bTracking THEN
						
						fHighestRecordedForce 	:= fForceInputABS;
						fLowestRecordedForce 	:= fForceInputABS;
						bTracking := TRUE;
						
					END_IF
						// Track max/min
					IF 	fDistance < fDisTanceSetPoint THEN
						IF fForceInputABS > fHighestRecordedForce THEN
							fHighestRecordedForce := fForceInputABS;
						END_IF;
			
						IF fForceInputABS < fLowestRecordedForce THEN
							fLowestRecordedForce  := fForceInputABS;
						END_IF;
					END_IF;
					
					
	//Evaluation
    ELSIF bEvaluate THEN
        
						bFail := (fHighestRecordedForce > fThreshold_UpperLimit) OR
      							 (fHighestRecordedForce  < fThreshold_LowerLimit);
						bPass := NOT bFail;
					
						bTracking := FALSE;
						bDistancePass := FALSE;					
    END_IF

ELSE
		// Clear 
		bPass 					:= FALSE;
		bFail 					:= FALSE;
		bOutOfRangeHigh 		:= FALSE;
		bOutOfRangeLow 			:= FALSE;
		fHighestRecordedForce 	:= 0.0;
		fLowestRecordedForce 	:= 0.0;
		bTracking 				:= FALSE;
		bActiveLast 			:= FALSE;
    	fForceLastStable 		:= 0.0;
    	fForceFiltered 			:= 0.0;
    	bForceStable 			:= FALSE;
		tonDebounce			 (IN:= FALSE);
END_IF

IF bReset THEN
		// Reset 
		bPass 					:= FALSE;
		bFail 					:= FALSE;
		bOutOfRangeHigh 		:= FALSE;
		bOutOfRangeLow 			:= FALSE;
		fHighestRecordedForce 	:= 0.0;
		fLowestRecordedForce 	:= 0.0;
		bTracking 				:= FALSE;
		bActiveLast 			:= FALSE;
    	fForceLastStable 		:= 0.0;
    	fForceFiltered 			:= 0.0;
    	bForceStable 			:= FALSE;
		tonDebounce			 (IN:= FALSE);
END_IF
//----------------------------------------------------------------------------oldschoo1

END_FUNCTION_BLOCK

// ---- POUs/03_Utilities/FB_DistanceMonitor.TcPOU
FUNCTION_BLOCK FB_DistanceMonitor
VAR_INPUT
    StartSignal   : BOOL;   // Signal indicating the start of the measurement cycle
    EndSignal     : BOOL;   // Signal indicating the end of the measurement cycle
	DistanceMaxSetpoint : BOOL;
    DistanceInput : REAL;   // Current distance reading
	fDistanceSetpoint: REAL;
END_VAR

VAR_OUTPUT
    MaxDistance   : REAL;   // Maximum distance during the cycle
    IsMeasuring   : BOOL;   // Flag indicating if the measurement cycle is active
	bDistancePass : BOOL;
	bDistanceFail : BOOL;
END_VAR

VAR
    CurrentMax    : REAL;   // Variable to hold the current maximum value during the cycle

END_VAR

// When StartSignal is triggered, initialize the measuring process


IF StartSignal AND NOT IsMeasuring THEN
    CurrentMax := DistanceInput; // Initialize the first measurement as the maximum
    IsMeasuring := TRUE;         // Set the measuring flag
	bDistancePass := FALSE;
	bDistanceFail := FALSE;
END_IF

// Monitor the maximum distance while the cycle is active
IF IsMeasuring THEN
    IF DistanceInput > CurrentMax THEN
        CurrentMax := DistanceInput;  // Update the maximum distance if a higher value is found
    END_IF
END_IF

// When EndSignal is triggered, finalize the measurement cycle and store the maximum value
IF EndSignal AND IsMeasuring THEN
    MaxDistance := CurrentMax;  // Store the maximum distance measured in the cycle
	IF MaxDistance > fDistanceSetpoint THEN
		bDistancePass		:= TRUE;
	ELSE bDistanceFail		:= TRUE;
	END_IF
    IsMeasuring := FALSE;       // Reset the measuring flag for the next cycle
END_IF

END_FUNCTION_BLOCK

// ---- POUs/03_Utilities/FB_UnpackByteToBoolArray.TcPOU
FUNCTION_BLOCK FB_UnpackByteToBoolArray
VAR_INPUT
	inputByte : BYTE;
END_VAR
VAR_IN_OUT
    outputBits : ARRAY[0..7]OF BOOL;
END_VAR
VAR
    idx : INT;
END_VAR
//-----------------------------oldschoo1

FOR idx := 0 TO 7 
DO
outputBits[idx] := (inputByte AND SHL(1, idx)) <> 0;
END_FOR
//------------------------------------------oldschoo1

END_FUNCTION_BLOCK

// ---- POUs/03_Utilities/FB_ArrayOfByte2Real.TcPOU
FUNCTION_BLOCK FB_ArrayOfByte2Real //Little Endian
VAR_INPUT
	arrBytes 						:ARRAY[0..3]OF BYTE; //[0]=LSB,[3]=MSB
END_VAR
VAR_OUTPUT
	rValue   						:REAL;
END_VAR
VAR
	pBytes   						:POINTER TO BYTE;
    pReal    						:POINTER TO REAL;
END_VAR
//-----------------------------------------------------------------oldschoo1

//Type-punning via pointers
pBytes := ADR(arrBytes[0]);
pReal := pBytes;
rValue := pReal^;
//-----------------------------------------------------------------oldschoo1

END_FUNCTION_BLOCK

// ---- POUs/03_Utilities/FB_Real2ArrayOfByte.TcPOU
FUNCTION_BLOCK FB_Real2ArrayOfByte //Little Endian
VAR_INPUT
	rValue   						:REAL;
END_VAR
VAR_OUTPUT
	arrBytes 						:ARRAY[0..3]OF BYTE;//[0]=LSB,[3]=MSB
END_VAR
VAR
	pReal  							:POINTER TO REAL;
    pBytes 							:POINTER TO BYTE;
    idx      						:INT;
END_VAR
//-----------------------------------------------------------------oldschoo1

//Type-punning via pointers
pReal := ADR(rValue);
pBytes := pReal;

FOR idx := 0 TO 3 DO arrBytes[idx] := pBytes[idx]; END_FOR
//-----------------------------------------------oldschoo1

END_FUNCTION_BLOCK

// ---- POUs/03_Utilities/FB_Byte_To_Bits.TcPOU
FUNCTION_BLOCK FB_Byte_To_Bits
VAR_INPUT
    fbReal2Byte : ARRAY[0..3] OF BYTE; // Array de bytes de entrada
END_VAR

VAR_OUTPUT
    Result : ARRAY[0..31] OF BOOL; // Array para almacenar los bits
END_VAR

VAR
    byteIndex : INT;      // Índice para iterar sobre los bytes
    bitIndex : INT;       // Índice para iterar sobre los bits dentro de cada byte
    shiftAmount : INT;    // Desplazamiento de bits
    shiftMask : BYTE;     // Máscara para cada bit
END_VAR

// Iterar sobre cada byte en fbRealPosition2Byte
FOR byteIndex := 0 TO 3 DO
    // Iterar sobre los 8 bits de cada byte
    FOR bitIndex := 0 TO 7 DO
        shiftAmount := 7 - bitIndex; // Shift a la izquierda para obtener los bits de 7 a 0
        shiftMask := LREAL_TO_BYTE( EXPT(2, shiftAmount));  // Generar la máscara de 2^shiftAmount
        
        // Extraer cada bit y almacenarlo en arrOutBits
        Result[byteIndex * 8 + bitIndex] := (fbReal2Byte[byteIndex] AND shiftMask) <> 0;
    END_FOR
END_FOR

END_FUNCTION_BLOCK

// ---- POUs/03_Utilities/FB_BytesToReal.TcPOU
FUNCTION_BLOCK FB_BytesToReal
VAR_INPUT
    inBytes : ARRAY[0..3] OF BYTE; // input in format IEEE-754
END_VAR

VAR_OUTPUT
    outReal : REAL; // Result 
END_VAR

VAR
    pReal : POINTER TO REAL;
    pByte : POINTER TO BYTE;
    i : INT;
END_VAR


pReal := ADR(outReal);
pByte := ADR(inBytes[0]);
(*
FOR i := 0 TO 3 DO
    pReal^[i] := pByte[i];
END_FOR*)

END_FUNCTION_BLOCK

// ---- POUs/03_Utilities/FUN_PackBoolArrayToByte.TcPOU
FUNCTION FUN_PackBoolArrayToByte 	:BYTE
VAR_INPUT
		 Input						:ARRAY[0..7]OF BOOL;
END_VAR
VAR
		 idx						:INT;
END_VAR
//-----------------------------------------------oldschoo1

FUN_PackBoolArrayToByte := 0;

FOR idx:= 0 TO 7 
DO 
FUN_PackBoolArrayToByte := FUN_PackBoolArrayToByte OR TO_BYTE(SHL(BOOL_TO_INT(Input[idx]), idx)); 
END_FOR
//--------------------------------------------------------------------------------------oldschoo1

END_FUNCTION

// ---- POUs/01_MODULES/SMAC/S_Master_SMAC.TcPOU
PROGRAM S_Master_SMAC
VAR	 
eState								: E_SmacState;
	
/////////////////////////////////////////////INITIALIZATION FUNCTION/////////////////////////////////////////////////////
	fbSmacInitialization_L							: FB_SmacInitialization;
	I_O_fbSmacInitialization_L						:ST_Phasing_Home;

	fbSmacInitialization_R							: FB_SmacInitialization;
	I_O_fbSmacInitialization_R						:ST_Phasing_Home;

/////////////////////////////////////////////CYCLE/MANUAL FUNCTION/////////////////////////////////////////////////////
	fbSmacCycleMan									: FB_SmacCycleMan;
	bTest											: BOOL;
/////////////////////////////////////////////CTRL SMAC/////////////////////////////////////////////////////
	nHomeState										: DINT;	
	nCyclePickState									: DINT;
	nCycleScrewkState								: DINT;
	nHomeStateManual								: DINT;	
	nCyclePickStateManual							: DINT;
	nCycleScrewkStateManual							: DINT;
	bLinealHomed									: BOOL;
	bRotativeHomed									: BOOL;
	bFirstCycle										: BOOL;
	
	
	aCycleFlag										: ARRAY[0..10] OF BOOL;

/////////////////////////////////////////////ERROR FUNCTION/////////////////////////////////////////////////////	
	fbErrorRST										: FB_ErrorReset;
	bEnbale_ErrorRST								: BOOL;
	bResetErrors									: BOOL;
	bAllErrorsCleared								: BOOL;
/////////////////////////////////////////////TIMERS / TRIGGERS/////////////////////////////////////////////////////
	tonResetError									:Tc2_Standard.TON;
	tonAbortModule									:Tc2_Standard.TON;
	tonCaseDelay									: ARRAY[0..40] OF TON;
	rTrigCase										: ARRAY[0..10] OF R_TRIG;
	CMDTrig											: ARRAY[0..10] OF R_TRIG;										
/////////////////////////////////////////////GRIPPERS CONTROL/////////////////////////////////////////////////////
	bCatchPiece							:BOOL;	//If set to TRUE - gripper OPEN || FALSE - gripper CLOSED
	bGuideScrew							:BOOL;	//If set to TRUE - gripper OPEN || FALSE - gripper CLOSED
	bGripperGuide_Timeout				:BOOL;	//Gripper didn't close in 3sec
	bGripperFixture_Timeout				:BOOL;	//Gripper didn't close in 3sec
	fbGripper_Guide						:FB_GripperCtrl;	
	fbGripper_Fixture					:FB_GripperCtrl;

END_VAR//---------------------------------------------------------------------------------------oldschoo1
VAR_OUTPUT
	stSmacReport						:ST_ProcessReport;
END_VAR

//--------------------IN/OUT----------------------------------------*
VAR_INPUT
	bCloseGripper						: BOOL;
	CMD									:ST_ModuleCMD;	
END_VAR
VAR_OUTPUT
	STATUS								:ST_ModuleStatus;
	I_O_fbSmacCycleMan					: ST_CYC_MAN;
END_VAR




//----------------------------------------------------------oldschoo1

PRG_Fault_SMAC(aAlarms := GVL_Master.stAlarms);
b_Ctrl_Smac();
c_FunctionProcess();
d_TimTrig();

ACTION a_StringDefinitions:

//////////////////////////////////////////STATUS STRING DEFINITIONS/////////////////////////////////////////////////////

	stSmacIO.sStatus[0]:='Initialization done';
	stSmacIO.sStatus[1]:='Servo enabled';
	stSmacIO.sStatus[2]:='';
	stSmacIO.sStatus[3]:='Motion execution acknowledge bit';
	stSmacIO.sStatus[4]:='Trajectory complete';
	stSmacIO.sStatus[5]:='';
	stSmacIO.sStatus[6]:='Homing Success';
	stSmacIO.sStatus[7]:='Homing failure';
	stSmacIO.sStatus[8]:='Phasing Succes';
	stSmacIO.sStatus[9]:='Phasing failure';
	stSmacIO.sStatus[10]:='Macro execution error';
	stSmacIO.sStatus[11]:='Macro execution';
	stSmacIO.sStatus[12]:='General fault';
	stSmacIO.sStatus[13]:='Servo error';
	stSmacIO.sStatus[14]:='STO fault';
	stSmacIO.sStatus[15]:='STO status';
	stSmacIO.sStatus[16]:='STO Input 1 de-energized';
	stSmacIO.sStatus[17]:='STO Input 2 de-energized';
	stSmacIO.sStatus[18]:='I2T fault';
	stSmacIO.sStatus[19]:='Driver overtemperature fault';
	stSmacIO.sStatus[20]:='Initialization done';
	
//////////////////////////////////////////MODE OF OPERATION STRING DEFINITIONS/////////////////////////////////////////////////////
	
	stSmacIO.sModeOfOperation[0] :='';
	stSmacIO.sModeOfOperation[1] :='Absolute position move';
	stSmacIO.sModeOfOperation[2] :='Relative position move';
	stSmacIO.sModeOfOperation[3] :='Velocity move';
	stSmacIO.sModeOfOperation[4] :='Torque move';
	stSmacIO.sModeOfOperation[5] :='Current move/QM1';
	stSmacIO.sModeOfOperation[6] :='Homing';
	stSmacIO.sModeOfOperation[7] :='Phasing';
	stSmacIO.sModeOfOperation[8] :='Current move/QM2';
	stSmacIO.sModeOfOperation[9] :='';
	stSmacIO.sModeOfOperation[10] :='Macro execution**';
	
//////////////////////////////////////////CONTRO WORD STRING DEFINITIONS/////////////////////////////////////////////////////

stSmacIO.sControlWord[0] :='';
stSmacIO.sControlWord[1] :='Start motion/macro start';
stSmacIO.sControlWord[2] :='Stop motion';
stSmacIO.sControlWord[3] :='Motor off';
stSmacIO.sControlWord[4] :='Motor on';
stSmacIO.sControlWord[5] :='Fault reset';
END_ACTION

ACTION b_Ctrl_Smac:

IF cmd.bAbort OR NOT stSafety.bSafety_OK OR NOT cmd.bEnable   THEN
	eState									:= E_SmacState.ABORTED;
END_IF

IF CMDTrig[4].Q THEN
	eState									:= E_SmacState.RESET_ERROR;
END_IF

IF eState = E_SmacState.MANUAL THEN
	I_O_fbSmacCycleMan.bManual_fbSmacCycleMan := TRUE;
ELSE I_O_fbSmacCycleMan.bManual_fbSmacCycleMan := FALSE;
END_IF

IF CMD.bManualMode THEN
	eState									:= E_SmacState.MANUAL;
END_IF
									

CMDTrig[0]( CLK := cmd.bAbort OR NOT stSafety.bSafety_OK OR NOT cmd.bEnable );
CMDTrig[1]( CLK := CMD.bEnable AND tonCaseDelay[3].Q );
CMDTrig[2]( CLK := CMD.bExecute);
CMDTrig[3]( CLK := CMD.bManualMode);
CMDTrig[4]( CLK := CMD.bReset);

		
(*******************************************************CTRL***********************************************************)
// Axis CTRL State Machine
CASE eState OF //--------------------------------------------------------------------------------------------------SM
	
E_SmacState.ABORTED://-------------------------------------------------------------------------------------------ABORTED:

						IF tonCaseDelay[22].Q THEN
							eState 												:= E_SmacState.ERROR;						
						END_IF

						IF  CMD.bEnable THEN
							eState 												:= E_SmacState.HOMING;
						END_IF
						//RESETTING
						I_O_fbSmacInitialization_R.bFunctionRequest				:= FALSE;
						I_O_fbSmacInitialization_L.bFunctionRequest				:= FALSE;
						I_O_fbSmacInitialization_R.bReset						:= TRUE;
						I_O_fbSmacInitialization_L.bReset						:= TRUE;
						I_O_fbSmacInitialization_L.bAcknowledge					:= FALSE;
						I_O_fbSmacInitialization_R.bAcknowledge					:= FALSE;
						
						I_O_fbSmacCycleMan.bAutoCycleRequest					:= FALSE;
						I_O_fbSmacCycleMan.bResetAutoCycle						:= TRUE;
						I_O_fbSmacCycleMan.bInitSecondPart						:= FALSE;
						I_O_fbSmacCycleMan.bAutoCycleAcknowledge				:= FALSE;
						aCycleFlag[1]											:= FALSE;
						aCycleFlag[2]											:= FALSE;
						aCycleFlag[3]											:= FALSE;
						
						nHomeState												:= 0;
						nCyclePickState											:= 0;
						nCycleScrewkState										:= 0;
						
						bCloseGripper											:= FALSE;
						
						IF tonCaseDelay[3].Q THEN
							I_O_fbSmacInitialization_R.bReset					:= FALSE;
							I_O_fbSmacInitialization_L.bReset					:= FALSE;
							I_O_fbSmacInitialization_R.bEnable					:= FALSE;
							I_O_fbSmacInitialization_L.bEnable					:= FALSE;
							
							I_O_fbSmacCycleMan.bResetAutoCycle					:= FALSE;
							I_O_fbSmacCycleMan.bCycProcess						:= FALSE;
							
							I_O_fbSmacCycleMan.bResetAutoCycle					:= FALSE;
							I_O_fbSmacCycleMan.bCycProcess						:= FALSE;
						END_IF
						

E_SmacState.HOMING://---------------------------------------------------------------------------------------------HOMING:
////////////////////////////////////////////////////LINEAL HOME////////////////////////////////////////////////////
						CASE 	nHomeState	OF
								
						0:
						IF aCycleFlag[1] THEN
							eState 												:= E_SmacState.AXIS_READY;
						ELSE nHomeState											:= 200;
						END_IF
						200:
						I_O_fbSmacInitialization_L.bEnable						:= TRUE;
						IF tonCaseDelay[6].Q THEN
							nHomeState											:= 300;
						END_IF
						300:
						I_O_fbSmacInitialization_L.bFunctionRequest				:= TRUE;
						IF tonCaseDelay[7].Q THEN
							nHomeState											:= 400;
						END_IF
						400:
						IF I_O_fbSmacInitialization_L.bAcknowledgeRequest THEN
							I_O_fbSmacInitialization_L.bAcknowledge				:= TRUE;
							nHomeState											:= 500;
							bLinealHomed										:= TRUE;
						ELSIF I_O_fbSmacInitialization_L.bPhasingError OR I_O_fbSmacInitialization_L.bHomeError THEN
							nHomeState											:= 500;
						END_IF
						500:
						I_O_fbSmacInitialization_L.bReset						:= TRUE;
						IF tonCaseDelay[8].Q THEN
							nHomeState											:= 600;
						END_IF
						600:
						I_O_fbSmacInitialization_L.bEnable						:= FALSE;
						I_O_fbSmacInitialization_L.bReset						:= FALSE;
						I_O_fbSmacInitialization_L.bFunctionRequest				:= FALSE;
						I_O_fbSmacInitialization_L.bAcknowledge					:= FALSE;
						IF bLinealHomed THEN
							nHomeState											:= 1200;
						END_IF
						
						1200:
						I_O_fbSmacInitialization_R.bEnable						:= TRUE;
						IF tonCaseDelay[9].Q THEN
							nHomeState											:= 1300;
						END_IF
						1300:
						I_O_fbSmacInitialization_R.bFunctionRequest				:= TRUE;
						IF tonCaseDelay[10].Q THEN
							nHomeState											:= 1400;
						END_IF
						1400:
						IF I_O_fbSmacInitialization_R.bAcknowledgeRequest THEN
							I_O_fbSmacInitialization_R.bAcknowledge				:= TRUE;
							nHomeState											:= 1500;
							bRotativeHomed										:= TRUE;
						ELSIF I_O_fbSmacInitialization_R.bPhasingError OR I_O_fbSmacInitialization_R.bHomeError THEN
							nHomeState											:= 1500;
						END_IF
						1500:
						I_O_fbSmacInitialization_R.bReset						:= TRUE;
						IF tonCaseDelay[11].Q THEN
							nHomeState											:= 1600;
						END_IF
						1600:
						I_O_fbSmacInitialization_R.bEnable						:= FALSE;
						I_O_fbSmacInitialization_R.bReset						:= FALSE;
						I_O_fbSmacInitialization_R.bFunctionRequest				:= FALSE;
						I_O_fbSmacInitialization_R.bAcknowledge					:= FALSE;
						IF bRotativeHomed AND bLinealHomed THEN
							bRotativeHomed										:= FALSE;
							bLinealHomed										:= FALSE;
							aCycleFlag[1]										:= TRUE;
							nHomeState											:= 0;
						END_IF
						
						5000://ERROR

						IF tonCaseDelay[12].Q THEN
							eState 												:= E_SmacState.ABORTED;
						END_IF
						END_CASE
	
						IF I_O_fbSmacInitialization_R.bHomeError OR I_O_fbSmacInitialization_R.bPhasingError OR
							I_O_fbSmacInitialization_L.bHomeError OR I_O_fbSmacInitialization_L.bPhasingError OR CMDTrig[0].Q THEN
							nHomeState											:= 5000;
						END_IF

		
E_SmacState.AXIS_READY://-------------------------------------------------------------------------------------AXIS_READY:
							
							aCycleFlag[1]										:= FALSE;
							aCycleFlag[3]										:= FALSE;
							//GO TO FIRST PART OF THE CYCLE
							IF (CMDTrig[2].Q AND stSmac.bSet_PickScrew) OR rTrigCase[1].Q THEN
									eState := E_SmacState.Cycle_Pick_Part;
							END_IF
										
							
E_SmacState.Cycle_Pick_Part://---------------------------------------------------------------------------Cycle_Pick_Part:		
							CASE nCyclePickState OF
							0:
							IF aCycleFlag[2] THEN
							eState 												:= E_SmacState.Cycle_Screw;
							ELSE nCyclePickState								:= 200;
							END_IF
							200:
							IF NOT bFirstCycle THEN
								nCyclePickState									:= 300;
							ELSE nCyclePickState								:= 400;
							END_IF
							300:
							I_O_fbSmacCycleMan.bSetValues						:= TRUE;
							IF tonCaseDelay[15].Q THEN
								nCyclePickState									:= 400;
							END_IF
							400:
							I_O_fbSmacCycleMan.bCycProcess						:= TRUE;
							IF tonCaseDelay[16].Q THEN
								nCyclePickState									:= 500;
							END_IF
							500:
							I_O_fbSmacCycleMan.bAutoCycleRequest				:= TRUE; 
							IF tonCaseDelay[17].Q THEN
								nCyclePickState									:= 600;
							END_IF
							600:
							IF I_O_fbSmacCycleMan.bFirstPartDoneFlag THEN
								aCycleFlag[2]									:= TRUE;
								nCyclePickState									:= 0;
							END_IF
							
							5000://ERROR
							IF tonCaseDelay[18].Q THEN
								eState 											:= E_SmacState.ABORTED;
							END_IF
							END_CASE
	
							IF I_O_fbSmacCycleMan.bCycError  THEN
								nCyclePickState										:= 5000;
							END_IF

						
							
							
E_SmacState.Cycle_Screw://-----------------------------------------------------------------------------------Cycle_Screw:
							aCycleFlag[2]										:= FALSE;
							CASE nCycleScrewkState OF
							0:	
							IF aCycleFlag[3] THEN//second part request
								eState 											:= E_SmacState.RECORD_CYCLE_DATA;
							ELSE nCycleScrewkState								:= 100;
							END_IF
							100:
							IF I_O_fbSmacCycleMan.bFirstPartDoneFlag AND CMDTrig[2].Q AND stSmac.bSet_ScrewItIn THEN
								I_O_fbSmacCycleMan.bInitSecondPart				:= TRUE;
								nCycleScrewkState								:= 200;
							END_IF
							200:
							bCloseGripper									:= I_O_fbSmacCycleMan.bOpenGuideGripper;
							IF I_O_fbSmacCycleMan.bAutoCycleAcknowledgeRequest THEN
								I_O_fbSmacCycleMan.bAutoCycleAcknowledge		:= TRUE;
								nCycleScrewkState								:= 300;
								
							END_IF
							300:
							IF I_O_fbSmacCycleMan.bCycleProcessDone THEN
								nCycleScrewkState								:= 400;
								I_O_fbSmacCycleMan.bAutoCycleAcknowledge		:= FALSE;
								I_O_fbSmacCycleMan.bAutoCycleRequest			:= FALSE;
								I_O_fbSmacCycleMan.bInitSecondPart				:= FALSE;
								I_O_fbSmacCycleMan.bSetValues					:= FALSE;
								I_O_fbSmacCycleMan.bResetAutoCycle				:= TRUE;
								nCycleScrewkState								:= 400;
							END_IF 
							400:
							IF tonCaseDelay[18].Q THEN
								I_O_fbSmacCycleMan.bResetAutoCycle				:= FALSE;
								I_O_fbSmacCycleMan.bCycProcess					:= FALSE;
								nCycleScrewkState								:= 500;
							END_IF
							500:
							nCycleScrewkState									:= 0;
							aCycleFlag[3]										:= TRUE;
							
							5000://ERROR
							IF tonCaseDelay[18].Q THEN
								eState 											:= E_SmacState.ABORTED;
							END_IF
							END_CASE
	
							IF I_O_fbSmacCycleMan.bCycError THEN
								nCycleScrewkState								:= 5000;
							END_IF

E_SmacState.RECORD_CYCLE_DATA://-----------------------------------------------------------------------------RECORD_CYCLE_DATA:

							
							stSmacReport.rSmac_Settings_LinearAcc				:= I_O_fbSmacCycleMan.nScaledLinearAcc;
							stSmacReport.rSmac_Settings_LinearVel				:= I_O_fbSmacCycleMan.nScaledLinearVel;
							stSmacReport.rSmac_Settings_LinearTorque			:= I_O_fbSmacCycleMan.nScaledLinearTorque;
							stSmacReport.rSmac_Settings_RotativeAcc				:= I_O_fbSmacCycleMan.nScaledRotativeAcc;
							stSmacReport.rSmac_Settings_RotativeVel				:= I_O_fbSmacCycleMan.nScaledRotativeVel;
							
							stSmacReport.bSmac_Pass								:= I_O_fbSmacCycleMan.bPass;
							stSmacReport.bSmac_Fail								:= I_O_fbSmacCycleMan.bFail;
				
							stSmacReport.rSmac_MaxDistanceReached				:= I_O_fbSmacCycleMan.MaxDistanceReached;
							IF tonCaseDelay[13].Q THEN
								eState 											:= E_SmacState.AXIS_READY;
 							END_IF
							

E_SmacState.RESET_ERROR://-----------------------------------------------------------------------------------------------ERROR:
							IF bAllErrorsCleared AND tonCaseDelay[4].Q THEN
								bEnbale_ErrorRST								:= FALSE;
							ELSE bEnbale_ErrorRST								:= TRUE;
							END_IF
							IF bFlash1Hz AND bEnbale_ErrorRST THEN
								bResetErrors									:= TRUE;
							ELSE bResetErrors									:= FALSE;
							END_IF
							IF tonCaseDelay[5].Q AND tonCaseDelay[4].Q THEN
								eState := E_SmacState.ABORTED;
							END_IF

E_SmacState.MANUAL://---------------------------------------------------------------------------------------------------MANUAL:
							IF NOT CMD.bManualMode THEN
								eState := E_SmacState.ABORTED;
							END_IF
							
ELSE 
eState := E_AxisState.ABORTED;
END_CASE //------------------------------------------------------------------------------------------------------END_CASE

(******************************************************STATUS************************************************************)
// Module Status
status.bReady					:= eState = E_SmacState.AXIS_READY;

status.bBusy					:= 	eState = E_SmacState.Cycle_Screw	OR
				   					eState = E_SmacState.Cycle_Pick_Part OR
				   					eState = E_SmacState.HOMING;
status.bFirstPartOfCycleDone	:=	I_O_fbSmacCycleMan.bFirstPartDoneFlag;	
		   
status.bDone					:= 	eState =	E_SmacState.RECORD_CYCLE_DATA;

status.bError					:= 	I_O_fbSmacInitialization_L.bHomeError OR I_O_fbSmacInitialization_R.bHomeError OR
								I_O_fbSmacInitialization_L.bPhasingError OR I_O_fbSmacInitialization_R.bPhasingError OR
								I_O_fbSmacCycleMan.bCycError OR stSmacIO.inStatusWordRotative.13 OR stSmacIO.inStatusWordLinear.13  ;
//--------------------------------------------------GRIPPERS-------------------------------------------------------------oldschoo1

IF CMD_Smac.bFixtureGripper OR (I_O_fbSmacCycleMan.bCloseFixtureGripper AND eState = E_AxisState.MANUAL_MODE) THEN
	bCatchPiece					:= TRUE;
ELSE bCatchPiece					:= FALSE;
END_IF

IF (CMD_Smac.bGuideGripper AND NOT bCloseGripper ) OR 
	(I_O_fbSmacCycleMan.bCloseGuideGripper AND eState = E_AxisState.MANUAL_MODE)THEN
	bGuideScrew					:= TRUE;
ELSE bGuideScrew					:= FALSE;
END_IF
END_ACTION

ACTION c_FunctionProcess:
//LINEAR PHASING AND HOME
fbSmacInitialization_L(	//INPUTS:
						bEnable 				:= I_O_fbSmacInitialization_L.bEnable,
						bAcknowledge 			:= I_O_fbSmacInitialization_L.bAcknowledge,
						bReset					:= I_O_fbSmacInitialization_L.bReset,
						bFunctionRequest		:= I_O_fbSmacInitialization_L.bFunctionRequest,
						nStatusWord				:= stSmacIO.inStatusWordLinear,
						nCurrentModeOfOperation	:= stSmacIO.inModeOfOperationLinear,							
						
						//OUTPUTS	
						bFunctionEnabled		=> I_O_fbSmacInitialization_L.bFunctionEnabled,
						bPhasingProcessDone		=> I_O_fbSmacInitialization_L.bPhasingProcessDone,
						bHomingProcessDone		=> I_O_fbSmacInitialization_L.bHomingProcessDone,
						bAcknowledgeRequest		=> I_O_fbSmacInitialization_L.bAcknowledgeRequest,
						bHomeError				=> I_O_fbSmacInitialization_L.bHomeError,
						bPhasingError			=> I_O_fbSmacInitialization_L.bPhasingError,
						//IN/OUT
						nControlWord			:= stSmacIO.qnControlWordLinear,								
						nModeOfOperation		:= stSmacIO.qnModeOfOperationLinear);
						
//ROTATIVE PHASING AND HOME						
fbSmacInitialization_R(	//INPUTS:
						bEnable 				:= I_O_fbSmacInitialization_R.bEnable,
						bAcknowledge 			:= I_O_fbSmacInitialization_R.bAcknowledge,
						bReset					:= I_O_fbSmacInitialization_R.bReset,
						bFunctionRequest		:= I_O_fbSmacInitialization_R.bFunctionRequest,
						nStatusWord				:= stSmacIO.inStatusWordRotative,
						nCurrentModeOfOperation	:= stSmacIO.inModeOfOperationRotative,							
						
						//OUTPUTS	
						bFunctionEnabled		=> I_O_fbSmacInitialization_R.bFunctionEnabled,
						bPhasingProcessDone		=> I_O_fbSmacInitialization_R.bPhasingProcessDone,
						bHomingProcessDone		=> I_O_fbSmacInitialization_R.bHomingProcessDone,
						bAcknowledgeRequest		=> I_O_fbSmacInitialization_R.bAcknowledgeRequest,
						bHomeError				=> I_O_fbSmacInitialization_R.bHomeError,
						bPhasingError			=> I_O_fbSmacInitialization_R.bPhasingError,
						//IN/OUT
						nControlWord			:= stSmacIO.qnControlWordRotative,								
						nModeOfOperation		:= stSmacIO.qnModeOfOperationRotative);
//CYCLE / MANUAL						
fbSmacCycleMan(			//INPUTS:
						nLinearVel				:= I_O_fbSmacCycleMan.nLinearVel,
						nLinearAcc				:= I_O_fbSmacCycleMan.nLinearAcc,
						nLinearSetPoint			:= I_O_fbSmacCycleMan.nLinearSetPoint,
						nLinearTorque			:= I_O_fbSmacCycleMan.nLinearTorque,
						bRotativeWorkPosition	:= I_O_fbSmacCycleMan.nRotativeWorkPosition,
						
						nRotativeVel			:= I_O_fbSmacCycleMan.nRotativeVel,
						nRotativeAcc			:= I_O_fbSmacCycleMan.nRotativeAcc,
						nRotativeSetPoint		:=  GVL_PERSISTENT.nSmacRotativeSetPoint,
						
						bCycProcess				:= I_O_fbSmacCycleMan.bCycProcess,
						bAutoCycleAcknowledge	:= I_O_fbSmacCycleMan.bAutoCycleAcknowledge,
						bAutoCycleRequest		:= I_O_fbSmacCycleMan.bAutoCycleRequest,
						bResetAutoCycle			:= I_O_fbSmacCycleMan.bResetAutoCycle,
						bInitSecondPart			:= I_O_fbSmacCycleMan.bInitSecondPart,
						bSetValues				:= GVL_HMI.bSmacSetValue OR (NOT bFirstCycle AND I_O_fbSmacCycleMan.bSetValues),
						bFixtureGripperClosed	:= stSmac.bGripperB_ClosedSensor,
						bGuideGripperClosed		:= stSmac.bGripperA_ClosedSensor,
						bManual					:= I_O_fbSmacCycleMan.bManual_fbSmacCycleMan,
						
						nDistanceSetPoint		:= I_O_fbSmacCycleMan.nDistanceSetPoint,				
						nDistanceTolerance		:= 500, //I_O_fbSmacCycleMan.nDistanceTolerance,
						bPickCycleMan			:= GVL_HMI.bSmacCyc1,
						bScrewCycleMan			:= GVL_HMI.bSmacCyc2,
						bHomeMan				:= GVL_HMI.bSmacHOME,
						//OUTPUTS
						bAutoCycleAcknowledgeRequest 	=> I_O_fbSmacCycleMan.bAutoCycleAcknowledgeRequest,
						bCycleProcessDone				=> I_O_fbSmacCycleMan.bCycleProcessDone,
						bFirstPartDoneFlag				=> I_O_fbSmacCycleMan.bFirstPartDoneFlag,
						bCycError						=> I_O_fbSmacCycleMan.bCycError,
						bOpenGuideGripper				=> I_O_fbSmacCycleMan.bOpenGuideGripper,
						bCloseGuideGripper				=> I_O_fbSmacCycleMan.bCloseGuideGripper,
						bCloseFixtureGripper			=> I_O_fbSmacCycleMan.bCloseFixtureGripper,
						bPass							=> I_O_fbSmacCycleMan.bPass,										
						bFail							=> I_O_fbSmacCycleMan.bFail,
						
						nScaledLinearVel				=> I_O_fbSmacCycleMan.nScaledLinearVel,			
						nScaledLinearAcc				=> I_O_fbSmacCycleMan.nScaledLinearAcc,						
						nScaledLinearSetPoint			=> I_O_fbSmacCycleMan.nScaledLinearSetPoint,						
						nScaledLinearTorque				=> I_O_fbSmacCycleMan.nScaledLinearTorque,					
	
						nScaledRotativeVel				=> I_O_fbSmacCycleMan.nScaledRotativeVel,						
						nScaledRotativeAcc				=> I_O_fbSmacCycleMan.nScaledRotativeAcc,					
						nScaledRotativeSetPoint			=> I_O_fbSmacCycleMan.nScaledRotativeSetPoint,
						MaxDistanceReached				=> I_O_fbSmacCycleMan.MaxDistanceReached,	
						bScrewAnimation					=> GVL_HMI.bScrewAnimation,
						//IN/OUT
						stSmacIO				:= stSmacIO);
						
							
									
												
//ERROR RESET
fbErrorRST(				//INPUTS
						bEnbale					:= bEnbale_ErrorRST,
						bResetErrors			:= bResetErrors,
						//OUTPUTS
						bAllErrorsCleared		=> bAllErrorsCleared,
						//IN/OUT
						stSmacIO				:= stSmacIO,
						bHomeError_L			:= I_O_fbSmacInitialization_L.bHomeError,
						bHomeError_R			:= I_O_fbSmacInitialization_R.bHomeError,
						bPhasingError_L			:= I_O_fbSmacInitialization_L.bPhasingError,
						bPhasingError_R			:= I_O_fbSmacInitialization_R.bPhasingError,
						bCycleError				:= I_O_fbSmacCycleMan.bCycError);

// Grippers CTRL
fbGripper_Fixture	 (bCloseGrip		:=bCatchPiece,
					  bClosedSensor		:=stSmac.bGripperB_ClosedSensor,
					  bOpen_Sig			=>stSmac.bGripperB_Open,
					  bClose_Sig		=>stSmac.bGripperB_Close,
					  bTimeout			=>bGripperFixture_Timeout);


fbGripper_Guide	     (bCloseGrip		:=bGuideScrew,
					  bClosedSensor		:=stSmac.bGripperA_ClosedSensor,
					  bOpen_Sig			=>(stSmac.bGripperA_Open ),
					  bClose_Sig		=>stSmac.bGripperA_Close,
					  bTimeout			=>bGripperGuide_Timeout);
END_ACTION

ACTION d_TimTrig:
//TIMERS

tonCaseDelay[0](IN := (eState =E_SmacState.HOMING) , PT := T#1S);
tonCaseDelay[1(*10*)](IN := eState = E_SmacState.Cycle_Screw , PT := T#1S);
tonCaseDelay[16](IN := eState = E_SmacState.Cycle_Pick_Part , PT := T#500MS);
tonCaseDelay[3](IN := (eState = E_SmacState.ABORTED) , PT := T#1S);
tonCaseDelay[4](IN := eState = E_SmacState.ERROR , PT := T#1S);
tonCaseDelay[13](IN := eState = E_SmacState.RECORD_CYCLE_DATA , PT := T#500MS);


tonCaseDelay[5](IN :=bAllErrorsCleared , PT := T#500MS);
tonCaseDelay[6](IN := nHomeState = 200 , PT := T#500MS);
tonCaseDelay[7](IN := nHomeState = 300 , PT := T#500MS);
tonCaseDelay[8](IN := nHomeState = 500 , PT := T#500MS);
tonCaseDelay[9](IN := nHomeState = 1200 , PT := T#500MS);
tonCaseDelay[10](IN := nHomeState = 1300 , PT := T#500MS);
tonCaseDelay[11](IN := nHomeState = 1500 , PT := T#500MS);
tonCaseDelay[12](IN := nHomeState = 5000 , PT := T#2S);

tonCaseDelay[15](IN := nCyclePickState = 300 , PT := T#500MS);
tonCaseDelay[16](IN := nCyclePickState = 400 , PT := T#500MS);  //??? the Same line 5
tonCaseDelay[17](IN := nCyclePickState = 500 , PT := T#500MS);
tonCaseDelay[18](IN := nCycleScrewkState = 400 , PT := T#500MS);


tonCaseDelay[21](IN := (stSmacIO.qnControlWordLinear = 2) , PT := T#1S);
tonCaseDelay[22](IN :=  stSmacIO.inStatusWordRotative.15 OR stSmacIO.inStatusWordRotative.16 OR
						 stSmacIO.inStatusWordRotative.17 OR stSmacIO.inStatusWordLinear.15 OR
						 stSmacIO.inStatusWordLinear.16 OR stSmacIO.inStatusWordLinear.17 
						, PT := T#500MS);

tonCaseDelay[23](IN :=cmd.bAbort OR NOT stSafety.bSafety_OK OR NOT cmd.bEnable , PT := T#1S);
tonCaseDelay[24](IN :=I_O_fbSmacCycleMan.bCycleProcessDone , PT := T#3S);


tonCaseDelay[26](IN := nHomeStatemanual = 200 , PT := T#500MS);
tonCaseDelay[27](IN := nHomeStatemanual = 300 , PT := T#500MS);
tonCaseDelay[28](IN := nHomeStatemanual = 500 , PT := T#500MS);
tonCaseDelay[29](IN := nHomeStatemanual = 1200 , PT := T#500MS);
tonCaseDelay[30](IN := nHomeStatemanual = 1300 , PT := T#500MS);
tonCaseDelay[31](IN := nHomeStatemanual = 1500 , PT := T#500MS);
tonCaseDelay[32](IN := nHomeStatemanual = 5000 , PT := T#2S);

tonCaseDelay[35](IN := nCyclePickStatemanual = 300 , PT := T#500MS);
tonCaseDelay[36](IN := nCyclePickStatemanual = 400 , PT := T#500MS);  //??? the Same line 5
tonCaseDelay[37](IN := nCyclePickStatemanual = 500 , PT := T#500MS);
tonCaseDelay[38](IN := nCycleScrewkStatemanual = 400 , PT := T#500MS);


//TRIGGERS
rTrigCase[0](CLK := eState = E_SmacState.ABORTED);
END_ACTION

END_PROGRAM

// ---- POUs/03_Utilities/SMAC/FB_SmacInitialization.TcPOU
FUNCTION_BLOCK FB_SmacInitialization
VAR_INPUT
	
	bEnable										: BOOL;
	bAcknowledge								: BOOL;
	bReset										: BOOL;
	bFunctionRequest							: BOOL;

END_VAR
VAR_OUTPUT
	
	bFunctionEnabled							: BOOL;
	bPhasingProcessDone							: BOOL;
	bHomingProcessDone							: BOOL;
	bAcknowledgeRequest							: BOOL;
	bHomeError									: BOOL;
	bPhasingError								: BOOL;

END_VAR
VAR
	nFunctionState								: DINT;
	sFunctionState								: STRING;
	tonCaseDelay								: ARRAY[0..10] OF TON;
	rTrigCase									: ARRAY[0..10] OF R_TRIG;
END_VAR
VAR_IN_OUT
	nStatusWord									: DINT;
	nControlWord								: UINT;
	nModeOfOperation							: UINT;
	nCurrentModeOfOperation						: DINT;
END_VAR

ACT_TimTrig();
IF bEnable THEN
	ACT_INIT();
	bFunctionEnabled 		:= TRUE;
ELSE bFunctionEnabled 		:= FALSE;
END_IF

ACTION ACT_INIT:
IF nStatusWord.13 THEN //ERROR
	nFunctionState := 5000;
ELSIF bReset THEN
	nFunctionState 					:= 0;
END_IF

CASE nFunctionState OF
	
0://Reset Values
bPhasingProcessDone				:= FALSE;
bHomingProcessDone				:= FALSE;
bAcknowledgeRequest				:= FALSE;
bHomeError						:= FALSE;
bPhasingError					:= FALSE;

IF bEnable AND NOT nStatusWord.15 AND NOT nStatusWord.16 AND NOT nStatusWord.17 THEN //STATUS 0 := MOTOR READY
	nFunctionState 				:= 15;
END_IF
15:
IF tonCaseDelay[8].Q THEN
	nFunctionState 				:= 20;
END_IF
20://home
sFunctionState 					:= 'Waiting Request';
IF rTrigCase[1].Q AND NOT nStatusWord.8 THEN
	nFunctionState 				:= 100;
ELSIF rTrigCase[1].Q AND  nStatusWord.8 THEN
nFunctionState 				:= 200;
END_IF

100://PHASING
sFunctionState 					:= 'Phasing Process';
IF tonCaseDelay[0].Q THEN
	nFunctionState 				:= 110;
END_IF
110://Resetting control word
nControlWord					:= 10;
nModeOfOperation				:= 7;
IF tonCaseDelay[1].Q AND (nCurrentModeOfOperation = 7) THEN
	nFunctionState 				:= 120;
END_IF
120://Setting control word
nControlWord					:= 1;
IF tonCaseDelay[2].Q  THEN
	nFunctionState 				:= 130;
END_IF
130://Phase done or error
IF tonCaseDelay[3].Q AND nStatusWord.8 THEN //STATUS 8 := PHASE DONE
	nFunctionState 				:= 200;
	bPhasingProcessDone 		:= TRUE;
ELSIF tonCaseDelay[3].Q AND nStatusWord.9 THEN //STATUS 8 := PHASE FAULT
	bPhasingError				:= TRUE;
	nFunctionState 				:= 5000;
END_IF


200: //HOMING
sFunctionState 					:= 'Homing Process';
IF tonCaseDelay[4].Q THEN
	nFunctionState 				:= 210;
END_IF
210://Resetting control word
nControlWord					:= 10;
nModeOfOperation				:= 6;
IF tonCaseDelay[5].Q AND (nCurrentModeOfOperation = 6) THEN
	nFunctionState 				:= 220;
END_IF
220://Setting control word
nControlWord					:= 1;
IF tonCaseDelay[6].Q THEN
	nFunctionState 				:= 230;
END_IF
230://Phase done or error
IF tonCaseDelay[7].Q AND nStatusWord.6 THEN //STATUS 8 := HOME DONE
	bHomingProcessDone	 		:= TRUE;
	nFunctionState 				:= 300;
ELSIF tonCaseDelay[7].Q AND nStatusWord.7 THEN //STATUS 8 := HOME FAULT
	nFunctionState 				:= 5000;
	bHomeError					:= TRUE;
END_IF
300://Process done, waiting acknowledge
sFunctionState 					:= 'Process done, Waiting for acknowledge';
bAcknowledgeRequest				:= TRUE;
IF bAcknowledge	THEN
	bAcknowledgeRequest			:= FALSE;
	nFunctionState 				:= 0;
END_IF
5000:
sFunctionState 					:= 'Error';
nModeOfOperation				:= 5;
IF bReset THEN
	nControlWord				:= 1;
ELSE nControlWord				:= 10;
END_IF
IF NOT nStatusWord.13 THEN
	nFunctionState 				:= 0;
END_IF


END_CASE
END_ACTION

ACTION ACT_TimTrig:
////////////////////////////////////////////TON///////////////////////////////////////////////////////
	tonCaseDelay[0](IN :=(nFunctionState = 100),PT := T#100MS);
	tonCaseDelay[1](IN :=(nFunctionState = 110),PT := T#100MS);
	tonCaseDelay[2](IN :=(nFunctionState = 120),PT := T#100MS);
	tonCaseDelay[3](IN :=(nFunctionState = 130),PT := T#100MS);
	tonCaseDelay[4](IN :=(nFunctionState = 200),PT := T#100MS);
	tonCaseDelay[5](IN :=(nFunctionState = 210),PT := T#100MS);
	tonCaseDelay[6](IN :=(nFunctionState = 220),PT := T#100MS);
	tonCaseDelay[7](IN :=(nFunctionState = 230),PT := T#100MS);
	tonCaseDelay[8](IN :=(nFunctionState = 15), PT := T#100MS);
	tonCaseDelay[9](IN :=, PT := T#100MS);
	
	
////////////////////////////////////////////TRIGGER///////////////////////////////////////////////////////
	rTrigCase[1](CLK := bFunctionRequest);
END_ACTION

END_FUNCTION_BLOCK

// ---- POUs/03_Utilities/SMAC/FB_SmacCycleMan.TcPOU
FUNCTION_BLOCK FB_SmacCycleMan

VAR_INPUT
	///////////////////////////////////////SETTINGS//////////////////////////////////////////////////
	nLinearVel						: DINT;
	nLinearAcc						: DINT;
	nLinearSetPoint					: DINT;
	nLinearTorque					: INT;
	
	nRotativeVel					: DINT;
	nRotativeAcc					: DINT;	
	nRotativeSetPoint				: DINT;//DINT;
		
	bFixtureGripperClosed			: BOOL;
	bGuideGripperClosed				: BOOL;

						 

///////////////////////////////////////MANUAL//////////////////////////////////////////////////
	bSetValues						: BOOL;
	bManual 						: BOOL;
	
	nManCycle						: DINT;
	bPickCycleMan					: BOOL;
	bScrewCycleMan					: BOOL;
	bHomeMan						: BOOL;
	
	

///////////////////////////////////////CYCLE//////////////////////////////////////////////////	
	bCycProcess						: BOOL;
	bAutoCycleAcknowledge			: BOOL;
	bAutoCycleRequest				: BOOL;
	bResetAutoCycle					: BOOL;
	bInitSecondPart					: BOOL;
	bRotativeWorkPosition			: DINT			:= 405;
	nUppperHeightLimit				: DINT;
	nLowerHeightLimit				: DINT;
///////////////////////////////////////REPORT//////////////////////////////////////////////////
	nDistanceSetPoint				: DINT;
	nDistanceTolerance				: DINT;
	
	
END_VAR
VAR_OUTPUT
	bAutoCycleAcknowledgeRequest	: BOOL;
	bCycleProcessDone				: BOOL;
	bFirstPartDoneFlag				: BOOL;
	bCycError						: BOOL;
	bOpenGuideGripper				: BOOL;
	bCloseGuideGripper				: BOOL;
	bCloseFixtureGripper			: BOOL;
	bPass							: BOOL;
	bFail							: BOOL;
	
	nScaledLinearVel				: DINT;
	nScaledLinearAcc				: DINT;
	nScaledLinearSetPoint			: DINT;
	nScaledLinearTorque				: INT;
	
	nScaledRotativeVel				: DINT;
	nScaledRotativeAcc				: DINT;	
	nScaledRotativeSetPoint			: DINT;
	
	MaxDistanceReached				: DINT;
	
	bScrewAnimation					: BOOL;
END_VAR
VAR
	tonCaseDelay					: ARRAY[0..40] OF TON;
	rTrigCase						: ARRAY[0..20] OF R_TRIG;
	bRotativeSetInPartPosition		: DINT			:= 405;
///////////////////////////////////////CYCLE//////////////////////////////////////////////////
	nCycleFunctionState				: DINT;
	bFirstAutoCycleFlag				: BOOL;
///////////////////////////////////////GENERAL//////////////////////////////////////////////////	
	bVelConst						: LREAL			:= 2621.44 ;
	bAccConst						: LREAL			:= 0.524288;
	bVelRotConst					: LREAL			:= 26214;
	

END_VAR
VAR_IN_OUT
	stSmacIO						: ST_SMAC_I_O;
END_VAR

IF bManual THEN
	ACT_Manual();
END_IF
IF bCycProcess	THEN
	ACT_Cycle();
END_IF

ACT_TimTrig();
ACT_Settings();

ACTION ACT_Cycle:
IF bResetAutoCycle  THEN
	nCycleFunctionState 				:= 0;	
END_IF

CASE nCycleFunctionState OF
	

0://HOMING
bFirstPartDoneFlag						:= FALSE;
bAutoCycleAcknowledgeRequest			:= FALSE;
bCycError								:= FALSE;
bScrewAnimation							:= FALSE;
stSmacIO.qnControlWordLinear 			:= 10;
stSmacIO.qnControlWordRotative			:= 10;
stSmacIO.qnModeOfOperationLinear		:= 4;
stSmacIO.qnModeOfOperationRotative		:= 2;
bOpenGuideGripper						:= FALSE;

IF rTrigCase[0].Q THEN
	nCycleFunctionState 				:= 20;
	bCycleProcessDone					:= FALSE;
	bPass								:= FALSE;
	bFail								:= FALSE;
END_IF

20:// CHECKING HOME AND PHASING
IF stSmacIO.inStatusWordLinear.6 AND stSmacIO.inStatusWordLinear.8 AND
	stSmacIO.inStatusWordRotative.6 AND stSmacIO.inStatusWordRotative.8 THEN
	nCycleFunctionState 				:= 200;
ELSE nCycleFunctionState 				:= 5000;
END_IF
200://SAFETY CHECK
IF (stSmacIO.inModeOfOperationLinear = 4) AND (stSmacIO.inModeOfOperationRotative = 2) AND
	NOT (stSmacIO.inStatusWordLinear.13) AND NOT (stSmacIO.inStatusWordRotative.13) AND
	(stSmacIO.inStatusWordLinear.1)AND (stSmacIO.inStatusWordRotative.1) THEN //else error
	nCycleFunctionState 				:= 300;
ELSE nCycleFunctionState 				:= 5000;
END_IF
300:
IF tonCaseDelay[11].Q THEN
	nCycleFunctionState 				:= 400;
END_IF
400://ROTATIVE TO WORK POSITION
stSmacIO.qnControlWordLinear 			:= 10;
stSmacIO.qnControlWordRotative 			:= 10;
stSmacIO.qnSetPointRotative 			:= bRotativeWorkPosition;
IF tonCaseDelay[12].Q THEN
	stSmacIO.qnControlWordRotative 		:= 1;
	nCycleFunctionState 				:= 450;
	
END_IF
450://ONCE ROTATIVE FINISH LINEAR START
IF tonCaseDelay[16].Q AND stSmacIO.inStatusWordRotative.4 THEN
	stSmacIO.qnControlWordLinear 		:= 1;
	nCycleFunctionState 				:= 500;
END_IF
500://linear get screw position 
IF tonCaseDelay[14].Q AND (stSmacIO.inCurrentPositionLinear > 8000(*it can change*)) THEN
	nCycleFunctionState 				:= 600;
	bScrewAnimation						:= TRUE;
END_IF
600://LINEAR SETTING TO GO TO HOME POSITION
stSmacIO.qnControlWordLinear 			:= 10;
stSmacIO.qnModeOfOperationLinear		:= 6;
IF tonCaseDelay[15].Q THEN
	nCycleFunctionState 				:= 700;
END_IF
700://LINEAR GO TO HOME POSITION
stSmacIO.qnControlWordLinear 			:= 1;
IF stSmacIO.inStatusWordLinear.4 THEN
	nCycleFunctionState 				:= 1000;
END_IF

1000: //WAITING SECOND PART
bFirstPartDoneFlag						:= TRUE;
IF rTrigCase[1].Q (*AND bFixtureGripperClosed	AND bGuideGripperClosed	*)THEN//Init second part
	nCycleFunctionState 				:= 1050;
END_IF
1050:
IF NOT (stSmacIO.inStatusWordLinear.13) AND NOT (stSmacIO.inStatusWordRotative.13) AND
	(stSmacIO.inStatusWordLinear.1)AND (stSmacIO.inStatusWordRotative.1) THEN //else errorTHEN //SECOND PART FLAG
	nCycleFunctionState 				:= 1100;
ELSE nCycleFunctionState 				:= 5000;
END_IF
1100: //SETTINGS SECOND PART
stSmacIO.qnSetVelocityRotative			:= 10; //RESETING VELOCITY
stSmacIO.qnControlWordLinear 			:= 10;
stSmacIO.qnControlWordRotative 			:= 10;
stSmacIO.qnModeOfOperationLinear		:= 4;
stSmacIO.qnSetPointRotative				:= bRotativeSetInPartPosition;//MOVEMENT TO SET IN PART
IF tonCaseDelay[17].Q THEN
	nCycleFunctionState 				:= 1200;
END_IF
1200: //START PROCESS
stSmacIO.qnSetVelocityRotative			:= nScaledRotativeVel; //SETTING VELOCITY
stSmacIO.qnControlWordLinear 			:= 1;
IF tonCaseDelay[18].Q THEN
	nCycleFunctionState 				:= 1300;
END_IF
1300: //WAITING FOR ROTATIVE
stSmacIO.qnControlWordRotative 			:= 1;
IF tonCaseDelay[19].Q AND stSmacIO.inStatusWordRotative.4 THEN
	nCycleFunctionState 				:= 1310;
END_IF
1310:
stSmacIO.qnControlWordRotative 			:= 10;
stSmacIO.qnSetPointRotative				:= nScaledRotativeSetPoint; 
IF tonCaseDelay[24].Q THEN
	nCycleFunctionState 				:= 1320;
END_IF
1320:
stSmacIO.qnControlWordRotative 			:= 1;
IF tonCaseDelay[25].Q  THEN
	nCycleFunctionState 				:= 1330;
END_IF
1330:
bOpenGuideGripper					:= TRUE;
IF tonCaseDelay[26].Q THEN
	nCycleFunctionState 				:= 1340;
END_IF
1340:
IF tonCaseDelay[28].Q AND tonCaseDelay[29].Q AND stSmacIO.inStatusWordRotative.4 THEN
	nCycleFunctionState 				:= 1360;
END_IF
1360:
MaxDistanceReached						:= stSmacIO.inCurrentPositionLinear;
IF tonCaseDelay[35].Q THEN
	nCycleFunctionState 				:= 1370;
	
END_IF
1370://it can be change by torque
IF MaxDistanceReached < nUppperHeightLimit AND
	MaxDistanceReached > nLowerHeightLimit THEN
	bPass								:= TRUE;
	bFail								:= FALSE;
ELSIF MaxDistanceReached > nUppperHeightLimit OR
	MaxDistanceReached < nLowerHeightLimit THEN
	bPass								:= FALSE;
	bFail								:= TRUE;
END_IF
IF tonCaseDelay[36].Q THEN
	nCycleFunctionState 					:= 1400;
END_IF

1400://SETTINGS TO GO HOME

stSmacIO.qnControlWordLinear 			:= 10;
stSmacIO.qnControlWordRotative 			:= 10;
stSmacIO.qnModeOfOperationLinear		:= 6;
stSmacIO.qnModeOfOperationRotative		:= 6;
IF tonCaseDelay[20].Q THEN
	nCycleFunctionState 				:= 1500;
END_IF
1500: //HOME POSITION
stSmacIO.qnControlWordLinear 			:= 1;
bScrewAnimation						:= FALSE;
IF tonCaseDelay[22].Q AND stSmacIO.inStatusWordLinear.4 THEN
	nCycleFunctionState 				:= 1600;
END_IF
1600://HOME PROCESS FINISH
stSmacIO.qnControlWordRotative 			:= 1;
IF tonCaseDelay[21].Q AND stSmacIO.inStatusWordRotative.4 THEN
	nCycleFunctionState 				:= 1700;
END_IF
1700://WAITING FOR ACKNOWLEDGE
bAutoCycleAcknowledgeRequest			:= TRUE;
IF bAutoCycleAcknowledge THEN
	bAutoCycleAcknowledgeRequest		:= FALSE;
	bCycleProcessDone					:= TRUE;
ELSIF tonCaseDelay[23].Q AND bAutoCycleAcknowledge THEN
	nCycleFunctionState 				:= 0;
END_IF

5000://CYCLE ERROR
bCycError								:= TRUE;
nCycleFunctionState 				:= 0;

END_CASE
END_ACTION

ACTION ACT_Manual:
IF tonCaseDelay[37].Q THEN
	nManCycle							:= 0;
END_IF

CASE nManCycle OF
0:
IF bPickCycleMan THEN
	nManCycle							:= 100;
ELSIF bScrewCycleMan THEN
	nManCycle							:= 1100;
ELSIF bHomeMan THEN
	nManCycle							:= 1900;
END_IF
stSmacIO.qnControlWordLinear 			:= 10;
stSmacIO.qnControlWordRotative			:= 10;
stSmacIO.qnModeOfOperationLinear		:= 4;
stSmacIO.qnModeOfOperationRotative		:= 2;

////////////////////////////////////////////////PICK CYCLE///////////////////////////////////////////////////////////////

100:// CHECKING HOME AND PHASING
IF stSmacIO.inStatusWordLinear.6 AND stSmacIO.inStatusWordLinear.8 AND
	stSmacIO.inStatusWordRotative.6 AND stSmacIO.inStatusWordRotative.8 THEN
	nManCycle 							:= 200;
ELSE nManCycle 							:= 5000;
END_IF
200://SAFETY CHECK
IF (stSmacIO.inModeOfOperationLinear = 4) AND (stSmacIO.inModeOfOperationRotative = 2) AND
	NOT (stSmacIO.inStatusWordLinear.13) AND NOT (stSmacIO.inStatusWordRotative.13) AND
	(stSmacIO.inStatusWordLinear.1)AND (stSmacIO.inStatusWordRotative.1) THEN //else error
	nManCycle 							:= 300;
ELSE nManCycle 							:= 5000;
END_IF
300:
IF tonCaseDelay[0].Q THEN
	nManCycle 							:= 400;
END_IF
400://ROTATIVE TO WORK POSITION
stSmacIO.qnSetPointRotative 			:= bRotativeWorkPosition;
IF tonCaseDelay[1].Q THEN
	stSmacIO.qnControlWordRotative 		:= 1;
	nManCycle 							:= 450;
	
END_IF
450://ONCE ROTATIVE FINISH LINEAR START
IF tonCaseDelay[2].Q AND stSmacIO.inStatusWordRotative.4 THEN
	stSmacIO.qnControlWordLinear 		:= 1;
	nManCycle 							:= 500;
END_IF
500:
IF tonCaseDelay[3].Q AND (stSmacIO.inCurrentPositionLinear > 8000) THEN
	nManCycle 							:= 600;
END_IF
600://LINEAR SETTING TO GO TO HOME POSITION
stSmacIO.qnControlWordLinear 			:= 10;
stSmacIO.qnModeOfOperationLinear		:= 6;
IF tonCaseDelay[4].Q THEN
	nManCycle 							:= 700;
END_IF
700://LINEAR GO TO HOME POSITION
stSmacIO.qnControlWordLinear 			:= 1;
IF stSmacIO.inStatusWordLinear.4 THEN
	nManCycle 							:= 0;
END_IF

////////////////////////////////////////////////SCREW CYCLE///////////////////////////////////////////////////////////////

1100:// CHECKING HOME AND PHASING
IF stSmacIO.inStatusWordLinear.6 AND stSmacIO.inStatusWordLinear.8 AND
	stSmacIO.inStatusWordRotative.6 AND stSmacIO.inStatusWordRotative.8 THEN
	nManCycle 							:= 1200;
ELSE nManCycle 							:= 5000;
END_IF
1200://SAFETY CHECK
IF (stSmacIO.inModeOfOperationLinear = 4) AND (stSmacIO.inModeOfOperationRotative = 2) AND
	NOT (stSmacIO.inStatusWordLinear.13) AND NOT (stSmacIO.inStatusWordRotative.13) AND
	(stSmacIO.inStatusWordLinear.1)AND (stSmacIO.inStatusWordRotative.1) THEN //else error
	nManCycle 							:= 1300;
ELSE nManCycle 							:= 5000;
END_IF
1300: 
bCloseGuideGripper						:= TRUE;
bCloseFixtureGripper					:= TRUE;
stSmacIO.qnSetVelocityRotative			:= 10; //RESETING VELOCITY
stSmacIO.qnSetPointRotative				:= bRotativeSetInPartPosition;//MOVEMENT TO SET IN PART
IF tonCaseDelay[5].Q THEN
	nManCycle 							:= 1400;
END_IF
1400: //START PROCESS
stSmacIO.qnSetVelocityRotative			:= nScaledRotativeVel; //SETTING VELOCITY
stSmacIO.qnControlWordLinear 			:= 1;
IF tonCaseDelay[6].Q THEN
	nManCycle 							:= 1500;
END_IF
1500: //WAITING FOR ROTATIVE
stSmacIO.qnControlWordRotative 			:= 1;
IF tonCaseDelay[7].Q AND stSmacIO.inStatusWordRotative.4 THEN
	nManCycle 							:= 1600;
END_IF
1600:
stSmacIO.qnControlWordRotative 			:= 10;
stSmacIO.qnSetPointRotative				:= nScaledRotativeSetPoint; 
IF tonCaseDelay[8].Q THEN
	nManCycle 							:= 1700;
END_IF
1700:
stSmacIO.qnControlWordRotative 			:= 1;
IF tonCaseDelay[9].Q  THEN
	nManCycle 							:= 1750;
END_IF
1750:

IF tonCaseDelay[31].Q THEN
	bCloseGuideGripper					:= FALSE;
	nManCycle 							:= 1800;
END_IF
1800:
IF  tonCaseDelay[29].Q AND stSmacIO.inStatusWordRotative.4 THEN
	nManCycle 							:= 1900;
END_IF
	
1900://SETTINGS TO GO HOME
stSmacIO.qnControlWordLinear 			:= 10;
stSmacIO.qnControlWordRotative 			:= 10;
stSmacIO.qnModeOfOperationLinear		:= 6;
stSmacIO.qnModeOfOperationRotative		:= 6;
IF tonCaseDelay[32].Q THEN
	nManCycle 							:= 2000;
END_IF
2000: //HOME POSITION
stSmacIO.qnControlWordLinear 			:= 1;
IF tonCaseDelay[33].Q AND stSmacIO.inStatusWordLinear.4 THEN
	nManCycle 							:= 2100;
	bCloseFixtureGripper				:= FALSE;
END_IF
2100://HOME PROCESS FINISH
stSmacIO.qnControlWordRotative 			:= 1;
IF tonCaseDelay[34].Q AND stSmacIO.inStatusWordRotative.4 THEN
	nManCycle							:= 0;
END_IF






END_CASE
END_ACTION

ACTION ACT_Settings:
//CONSTANTS IN BASE TO THE MANUAL

nScaledLinearVel 		:=LREAL_TO_DINT( bVelConst *nLinearVel);
nScaledLinearAcc 		:=LREAL_TO_DINT( bAccConst *nLinearAcc);
nDistanceSetPoint		:=REAL_TO_DINT( 200 *nLinearSetPoint);//6761
nScaledLinearSetPoint	:=10000;
nScaledLinearTorque		:=REAL_TO_INT( nLinearTorque*1365);

nScaledRotativeVel 		:=LREAL_TO_DINT( bVelConst *nRotativeVel);
nScaledRotativeAcc 		:=LREAL_TO_DINT( bAccConst *nRotativeAcc);
nScaledRotativeSetPoint	:=REAL_TO_DINT( 5.5 *nRotativeSetPoint);


IF rTrigCase[2].Q THEN	
	stSmacIO.qnSetVelocityLinear			:= nScaledLinearVel;
	stSmacIO.qnSetAcceleraionLinear			:= nScaledLinearAcc;
	stSmacIO.qnSetPointLinear				:= nScaledLinearSetPoint;
	stSmacIO.qnSetMaxiumTorqueLinear		:= nScaledLinearTorque;
	
	stSmacIO.qnSetVelocityRotative			:= nScaledRotativeVel;
	stSmacIO.qnSetAcceleraionRotative		:= nScaledRotativeAcc;
	stSmacIO.qnSetPointRotative				:= nScaledRotativeSetPoint;
	
END_IF

nUppperHeightLimit 							:= nDistanceSetPoint + nDistanceTolerance;
nLowerHeightLimit							:= nDistanceSetPoint - nDistanceTolerance;
END_ACTION

ACTION ACT_TimTrig:
	////////////////////////////////////////////TON//////////////////////////////////////////

	//MANUAL
	tonCaseDelay[0](IN :=nManCycle = 300,PT:= T#100MS ); 
	tonCaseDelay[1](IN :=nManCycle = 400,PT:= T#500MS );
	tonCaseDelay[2](IN :=nManCycle = 450,PT:= T#500MS );
	
	tonCaseDelay[3](IN := nManCycle = 500,PT:= T#100MS ); 
	tonCaseDelay[4](IN := nManCycle = 600,PT:= T#500MS );
	tonCaseDelay[5](IN := nManCycle = 1300,PT:= T#100MS );
	tonCaseDelay[6](IN := nManCycle = 1400,PT:= T#100MS );
	tonCaseDelay[7](IN := nManCycle = 1500,PT:= T#100MS );
	tonCaseDelay[8](IN := nManCycle = 1600,PT:= T#100MS );
	tonCaseDelay[9](IN := nManCycle = 1700,PT:= T#100MS );
	tonCaseDelay[31](IN := nManCycle = 1750,PT:= T#2S );
	tonCaseDelay[32](IN := nManCycle = 1900,PT:= T#500MS );
	tonCaseDelay[33](IN := nManCycle = 2000,PT:= T#500MS );
	tonCaseDelay[34](IN := nManCycle = 2100,PT:= T#500MS );
	//CYCLE
	tonCaseDelay[10](IN := nCycleFunctionState =10,PT:= T#100MS ); 
	tonCaseDelay[11](IN := nCycleFunctionState =300,PT:= T#100MS ); 
	tonCaseDelay[12](IN := nCycleFunctionState =400,PT:= T#500MS );
	tonCaseDelay[13](IN := nCycleFunctionState =150,PT:= T#500MS );
	tonCaseDelay[14](IN := nCycleFunctionState =500,PT:= T#1500MS );
	tonCaseDelay[15](IN := nCycleFunctionState =600,PT:= T#100MS );
	tonCaseDelay[16](IN := nCycleFunctionState =450,PT:= T#1S );
	tonCaseDelay[17](IN := nCycleFunctionState =1100,PT:= T#100MS );
	tonCaseDelay[18](IN := nCycleFunctionState =1200,PT:= T#1500MS );
	tonCaseDelay[19](IN := nCycleFunctionState =1300,PT:= T#1S );
	tonCaseDelay[20](IN := nCycleFunctionState =1400,PT:= T#100MS );
	tonCaseDelay[21](IN := nCycleFunctionState =1600 ,PT:= T#1S );
	tonCaseDelay[22](IN := nCycleFunctionState =1500,PT:= T#1S );
	tonCaseDelay[23](IN :=bAutoCycleAcknowledge ,PT:= T#1S );
	tonCaseDelay[24](IN :=nCycleFunctionState =1310 ,PT:= T#500MS );
	tonCaseDelay[25](IN := nCycleFunctionState =1320 ,PT:= T#500MS );
	tonCaseDelay[26](IN := NOT bGuideGripperClosed,PT:= T#1S );
	tonCaseDelay[27](IN :=nCycleFunctionState =1800,PT:= T#1S );
	tonCaseDelay[28](IN := nCycleFunctionState =1340 ,PT:= T#1S );
	tonCaseDelay[29](IN := stSmacIO.inStatusWordRotative.4 ,PT:= T#2S );
	tonCaseDelay[30](IN := nCycleFunctionState =1700,PT:= T#100MS );
	tonCaseDelay[35](IN := nCycleFunctionState =1360,PT:= T#500MS );
	tonCaseDelay[36](IN := nCycleFunctionState =1370,PT:= T#500MS );
	
	tonCaseDelay[37](IN := nManCycle <> 0,PT:= T#20S );
////////////////////////////////////////////TRIGGER//////////////////////////////////////////	
	rTrigCase[0]( CLK := bAutoCycleRequest);
	rTrigCase[1]( CLK := bInitSecondPart);
	rTrigCase[2]( CLK := bSetValues);
END_ACTION

END_FUNCTION_BLOCK

// ---- POUs/03_Utilities/SMAC/FB_ErrorReset.TcPOU
FUNCTION_BLOCK FB_ErrorReset
VAR_INPUT
	bEnbale							: BOOL;
	bResetErrors					: BOOL;
END_VAR
VAR_OUTPUT
	bAllErrorsCleared				: BOOL;
END_VAR
VAR
	tonCaseDelay									: ARRAY[0..10] OF TON;
	rTrigCase										: ARRAY[0..10] OF R_TRIG;
END_VAR
VAR_IN_OUT
	stSmacIO						: ST_SMAC_I_O;
	bHomeError_L					: BOOL;
	bHomeError_R					: BOOL;
	bPhasingError_L					: BOOL;
	bPhasingError_R					: BOOL;
	bCycleError						: BOOL;
	
	
END_VAR

IF bEnbale THEN
	ACT_ErrorReset();
END_IF

ACTION ACT_ErrorReset:
IF bResetErrors THEN
	
	bHomeError_L							:= FALSE;				
	bHomeError_R							:= FALSE;
	bPhasingError_L							:= FALSE;
	bPhasingError_R							:= FALSE;
	bCycleError								:= FALSE;

stSmacIO.qnControlWordLinear				:= 5;

IF tonCaseDelay[0].Q THEN
	stSmacIO.qnControlWordRotative				:= 5;
END_IF


IF (bHomeError_L				= FALSE) AND 
	(bHomeError_R				= FALSE) AND
	(bPhasingError_L			= FALSE) AND
	(bPhasingError_R			= FALSE) AND
	(bCycleError				= FALSE) AND NOT
	stSmacIO.inStatusWordLinear.13		 AND NOT
	stSmacIO.inStatusWordRotative.13	 THEN
	bAllErrorsCleared			:= TRUE;
ELSE bAllErrorsCleared			:= FALSE;
END_IF
END_IF
END_ACTION

ACTION ACT_TimTrig:
//TIMERS
	tonCaseDelay[0](IN := stSmacIO.qnControlWordLinear	= 5, PT:= T#500MS);
END_ACTION

END_FUNCTION_BLOCK

// ---- POUs/03_Utilities/FB_GripperCtrl.TcPOU
FUNCTION_BLOCK FB_GripperCtrl
VAR_INPUT
	
	bCloseGrip					:BOOL;
	bClosedSensor				:BOOL;

END_VAR
VAR_OUTPUT
	
	bOpen_Sig					:BOOL;
	bClose_Sig					:BOOL;
	bTimeout					:BOOL;

END_VAR
VAR
	tonOpenPulse				:Tc2_Standard.TON:=(PT:=T#1S);
	tonClosePulse				:Tc2_Standard.TON:=(PT:=T#1S);
	tonResetSignal				:ARRAY [1..2] OF Tc2_Standard.TON;
	tonTimeout					:Tc2_Standard.TON:=(PT:=T#3S);
	
END_VAR
//-------------------------------------------------------------------oldschoo1

//Timers
		 tonOpenPulse (IN:= NOT bCloseGrip);
		tonClosePulse (IN:= bCloseGrip);
		
	tonResetSignal[1] (IN:= NOT bCloseGrip,PT:=T#100MS);
	tonResetSignal[2] (IN:= bCloseGrip,PT:=T#100MS);
	
		   tonTimeout (IN:= bClose_Sig AND NOT bClosedSensor);

// Logic
IF NOT bCloseGrip THEN //-----------------------------------------------KEEP_OPEN

								bClose_Sig 		:= FALSE;
						
						IF tonResetSignal[1].Q 
							THEN	
								bOpen_Sig 		:= TRUE;
						END_IF							
ELSE //----------------------------------------------------------------CLOSE_GRIP
	
								bOpen_Sig 		:= FALSE;
						
							IF tonResetSignal[2].Q 
							THEN	
								bClose_Sig 		:= TRUE;
						END_IF										
END_IF
bTimeout := tonTimeout.Q; //----------------------------------------------TIMEOUT

//-----------------------------------------------------------------------oldschoo1

END_FUNCTION_BLOCK

// ---- POUs/01_MODULES/SMAC/PRG_Fault_SMAC.TcPOU
PROGRAM PRG_Fault_SMAC
VAR
	i					: INT;
	bTest				: BOOL;
END_VAR
VAR_IN_OUT
  aAlarms  : ARRAY[0..3] OF ST_Events;
END_VAR

IF GVL_PERSISTENT.bSMACEnable THEN 
ACT_FaultTrig();
END_IF

(************************************** Faults reset **********************************************)
IF   bResetButtonRisingEdge THEN 
	FOR i := 0 TO 127 DO
		GVL_MASTER.stAlarms[3].aEventFlags[i] := FALSE;
	END_FOR
END_IF
//===============================================================
//Initialize event texts on first scan
IF NOT GVL_MASTER.stAlarms[3].bEventTextsSet THEN
	SetEventTexts();
	GVL_MASTER.stAlarms[3].bEventTextsSet := TRUE;
END_IF


(***************************************************************************************************)
//Immediate fault
GVL_MASTER.stAlarms[3].bImmediateFault := FALSE;
FOR i := 0 TO 32DO
	GVL_MASTER.stAlarms[3].bImmediateFault := GVL_MASTER.stAlarms[3].bImmediateFault OR GVL_MASTER.stAlarms[3].aEventFlags[i];
END_FOR

//Cycle stop fault
GVL_MASTER.stAlarms[3].bCycleStopFault := FALSE;
FOR i := 33 TO 79 DO
	GVL_MASTER.stAlarms[3].bCycleStopFault := GVL_MASTER.stAlarms[3].bCycleStopFault OR GVL_MASTER.stAlarms[3].aEventFlags[i];
END_FOR

//Cycle stop REQUEST
GVL_MASTER.stAlarms[3].bCycleStopRequest := FALSE;
FOR i := 80 TO 99 DO
	GVL_MASTER.stAlarms[3].bCycleStopRequest := GVL_MASTER.stAlarms[3].bCycleStopRequest OR GVL_MASTER.stAlarms[3].aEventFlags[i];
END_FOR

ACTION ACT_FaultTrig:

//Station 3 - SMAC Linear Servo error
IF stSmacIO.inStatusWordLinear.13 THEN 
	stAlarms[3].aEventFlags[2] := TRUE;
	bTest							:= TRUE;
END_IF
//Station 3 - SMAC Rotative Servo error
IF stSmacIO.inStatusWordRotative.13 THEN 
	stAlarms[3].aEventFlags[4] := TRUE;
	bTest							:= TRUE;
END_IF
//Station 3 - SMAC STO Fault
IF stSmacIO.inStatusWordRotative.15 OR stSmacIO.inStatusWordLinear.15 THEN 
	stAlarms[3].aEventFlags[5] := TRUE;
	bTest							:= TRUE;
END_IF
//Station 3 - SMAC I2T Fault
IF stSmacIO.inStatusWordRotative.18 OR stSmacIO.inStatusWordLinear.18 THEN 
	stAlarms[3].aEventFlags[6] := TRUE;
	bTest							:= TRUE;
END_IF
//Station 3 - SMAC Over temperature Fault
IF stSmacIO.inStatusWordRotative.19 OR stSmacIO.inStatusWordLinear.19 THEN 
	stAlarms[3].aEventFlags[7] := TRUE;
	bTest							:= TRUE;
END_IF




